(* PLC project Adressering.ecp, WAGO e!COCKPIT e!COCKPIT *)
(* stored: creationDateTime 2021-01-18T14:20:23.2110188, modificationDateTime 2021-01-18T11:51:27.6823754 *)

TYPE dtRomtype_99999 : STRUCT
  RB601_V : BOOL;  (* Bevegelse *)
  RB602_V : BOOL;  (* Bevegelse *)
  RB603_V : BOOL;  (* Bevegelse *)
  RB604_V : BOOL;  (* Bevegelse *)
  RB605_V : BOOL;  (* Bevegelse *)
  RB606_V : BOOL;  (* Bevegelse *)
  RB607_V : BOOL;  (* Bevegelse *)
  RB608_V : BOOL;  (* Bevegelse *)
  RB609_V : BOOL;  (* Bevegelse *)
  RB601_HVAC : BOOL;  (* HVAC signal *)
  RB602_HVAC : BOOL;  (* HVAC signal *)
  RB603_HVAC : BOOL;  (* HVAC signal *)
  RB604_HVAC : BOOL;  (* HVAC signal *)
  RB605_HVAC : BOOL;  (* HVAC signal *)
  RB606_HVAC : BOOL;  (* HVAC signal *)
  RB607_HVAC : BOOL;  (* HVAC signal *)
  RB608_HVAC : BOOL;  (* HVAC signal *)
  RB609_HVAC : BOOL;  (* HVAC signal *)
  RT601_CT : REAL;  (* Rom temperatur *)
  RT602_CT : REAL;  (* Rom temperatur *)
  RT602_SP : REAL;  (* Temperatur SP *)
  RT603_CT : REAL;  (* Rom temperatur *)
  RT603_SP : REAL;  (* Temperatur SP *)
  RT604_CT : REAL;  (* Rom temperatur *)
  RT604_SP : REAL;  (* Temperatur SP *)
  RT605_CT : REAL;  (* Rom temperatur *)
  RT605_SP : REAL;  (* Temperatur SP *)
  RT606_CT : REAL;  (* Rom temperatur *)
  RT606_SP : REAL;  (* Temperatur SP *)
  RT607_CT : REAL;  (* Rom temperatur *)
  RT607_SP : REAL;  (* Temperatur SP *)
  RT608_CT : REAL;  (* Rom temperatur *)
  RT608_SP : REAL;  (* Temperatur SP *)
  RT609_CT : REAL;  (* Rom temperatur *)
  RT609_SP : REAL;  (* Temperatur SP *)
  RT601_SP_D : REAL;  (* Temperatur SP *)
  RT601_SP_S : REAL;  (* Temperatur SP standby *)
  RT601_SP_N : REAL;  (* Temperatur SP nattsenk *)
  RT601_SP_F : REAL;  (* Temperatur SP frostsikring *)
  RT601_CS : REAL;  (* Aktivt temperatur SP *)
  OPM : INT;  (* Rom modus *)
  OPM_CV : INT;  (* Rom modus verdi *)
  RY601_CV : REAL;  (* Co2 Nivaa *)
  RY602_CV : REAL;  (* Co2 Nivaa *)
  RY603_CV : REAL;  (* Co2 Nivaa *)
  RY604_CV : REAL;  (* Co2 Nivaa *)
  RY605_CV : REAL;  (* Co2 Nivaa *)
  RY606_CV : REAL;  (* Co2 Nivaa *)
  RY607_CV : REAL;  (* Co2 Nivaa *)
  RY608_CV : REAL;  (* Co2 Nivaa *)
  RY609_CV : REAL;  (* Co2 Nivaa *)
  RY601_SP : REAL;  (* Co2 SP *)
  RY601_MAN : BOOL;  (* Co2 Man mode *)
  RY601_OP : REAL;  (* Co2 paadrag *)
  LH601_OP : REAL;  (* Varmepaadrag *)
  LH602_OP : REAL;  (* Varmepaadrag *)
  LH603_OP : REAL;  (* Varmepaadrag *)
  LH604_OP : REAL;  (* Varmepaadrag *)
  LH605_OP : REAL;  (* Varmepaadrag *)
  LH606_OP : REAL;  (* Varmepaadrag *)
  LH607_OP : REAL;  (* Varmepaadrag *)
  LH608_OP : REAL;  (* Varmepaadrag *)
  LH609_OP : REAL;  (* Varmepaadrag *)
  LH601_MAN : BOOL;  (* Force LH *)
END_STRUCT;
END_TYPE

TYPE dtRomtype_9992 : STRUCT
  RB601_V : BOOL;  (* Bevegelse *)
  RB602_V : BOOL;  (* Bevegelse *)
  RB603_V : BOOL;  (* Bevegelse *)
  RB604_V : BOOL;  (* Bevegelse *)
  RB605_V : BOOL;  (* Bevegelse *)
  RB606_V : BOOL;  (* Bevegelse *)
  RB607_V : BOOL;  (* Bevegelse *)
  RB608_V : BOOL;  (* Bevegelse *)
  RB609_V : BOOL;  (* Bevegelse *)
  RB601_HVAC : BOOL;  (* HVAC signal *)
  RB602_HVAC : BOOL;  (* HVAC signal *)
  RB603_HVAC : BOOL;  (* HVAC signal *)
  RB604_HVAC : BOOL;  (* HVAC signal *)
  RB605_HVAC : BOOL;  (* HVAC signal *)
  RB606_HVAC : BOOL;  (* HVAC signal *)
  RB607_HVAC : BOOL;  (* HVAC signal *)
  RB608_HVAC : BOOL;  (* HVAC signal *)
  RB609_HVAC : BOOL;  (* HVAC signal *)
  RT601_CT : REAL;  (* Rom temperatur *)
  RT602_CT : REAL;  (* Rom temperatur *)
  RT602_SP : REAL;  (* Temperatur SP *)
  RT603_CT : REAL;  (* Rom temperatur *)
  RT603_SP : REAL;  (* Temperatur SP *)
  RT604_CT : REAL;  (* Rom temperatur *)
  RT604_SP : REAL;  (* Temperatur SP *)
  RT605_CT : REAL;  (* Rom temperatur *)
  RT605_SP : REAL;  (* Temperatur SP *)
  RT606_CT : REAL;  (* Rom temperatur *)
  RT606_SP : REAL;  (* Temperatur SP *)
  RT607_CT : REAL;  (* Rom temperatur *)
  RT607_SP : REAL;  (* Temperatur SP *)
  RT608_CT : REAL;  (* Rom temperatur *)
  RT608_SP : REAL;  (* Temperatur SP *)
  RT609_CT : REAL;  (* Rom temperatur *)
  RT609_SP : REAL;  (* Temperatur SP *)
  RT601_SP_D : REAL;  (* Temperatur SP *)
  RT601_SP_S : REAL;  (* Temperatur SP standby *)
  RT601_SP_N : REAL;  (* Temperatur SP nattsenk *)
  RT601_SP_F : REAL;  (* Temperatur SP frostsikring *)
  RT601_CS : REAL;  (* Aktivt temperatur SP *)
  OPM : INT;  (* Rom modus *)
  OPM_CV : INT;  (* Rom modus verdi *)
  RY601_CV : REAL;  (* Co2 Nivaa *)
  RY602_CV : REAL;  (* Co2 Nivaa *)
  RY601_SP : REAL;  (* Co2 SP *)
  RY601_MAN : BOOL;  (* Co2 Man mode *)
  RY601_OP : REAL;  (* Co2 paadrag *)
END_STRUCT;
END_TYPE

TYPE dtRomtype_111001 : STRUCT
  RB601_V : BOOL;  (* Bevegelse *)
  RB601_HVAC : BOOL;  (* HVAC signal *)
  RT601_CT : REAL;  (* Rom temperatur *)
  RT601_SP_D : REAL;  (* Temperatur SP *)
  RT601_SP_S : REAL;  (* Temperatur SP standby *)
  RT601_SP_N : REAL;  (* Temperatur SP nattsenk *)
  RT601_SP_F : REAL;  (* Temperatur SP frostsikring *)
  RT601_CS : REAL;  (* Aktivt temperatur SP *)
  OPM : INT;  (* Rom modus *)
  OPM_CV : INT;  (* Rom modus verdi *)
  LH601_CMD : BOOL;  (* LH601_CMD *)
  LH601_MAN : BOOL;  (* Force LH *)
END_STRUCT;
END_TYPE

TYPE dtRomtype_111111111111111 : STRUCT
  RB601_V : BOOL;  (* Bevegelse *)
  RB601_HVAC : BOOL;  (* HVAC signal *)
  RT601_CT : REAL;  (* Rom temperatur *)
  RT601_SP_D : REAL;  (* Temperatur SP *)
  RT601_SP_S : REAL;  (* Temperatur SP standby *)
  RT601_SP_N : REAL;  (* Temperatur SP nattsenk *)
  RT601_SP_F : REAL;  (* Temperatur SP frostsikring *)
  RT601_CS : REAL;  (* Aktivt temperatur SP *)
  OPM : INT;  (* Rom modus *)
  OPM_CV : INT;  (* Rom modus verdi *)
  RY601_CV : REAL;  (* Co2 Nivaa *)
  RY601_SP : REAL;  (* Co2 SP *)
  RY601_MAN : BOOL;  (* Co2 Man mode *)
  RY601_OP : REAL;  (* Co2 paadrag *)
  LH601_OP : REAL;  (* Varmepaadrag *)
  LH601_MAN : BOOL;  (* Force LH *)
  LH601_CMD : BOOL;  (* LH601_CMD *)
  LC601_OP : REAL;  (* LC601_OP *)
  LC601_SP : REAL;  (* LC SP *)
  LC601_MAN : BOOL;  (* Force LC *)
  LC601_CMD : BOOL;  (* LC601_CMD *)
  RT601_SP : REAL;  (* Temperatur SP feedback *)
  RT601_SP_FB : REAL;  (* Temperatur SP *)
  RT601_SP_IN : REAL;  (* Temperatur SP lokalt panel *)
  LU601_V : BOOL;  (* Befukter status *)
  LU601_AL : BOOL;  (* Befukter alarm/feil *)
  LU601_CMD : BOOL;  (* Befukter tillat start *)
  OPM_001 : BYTE;  (* OPM output *)
  RH601 : REAL;  (* Rom fuktighet *)
END_STRUCT;
END_TYPE

{attribute 'qualified_only'}
VAR_GLOBAL  (* STLV59_563 *)
  STLV59_A_563_RB001_HVAC : BOOL;  (* HVAC signal for PLS *)
  STLV59_A_563_KNX_Card_1_Status : BOOL;  (* KNX kort 1 status *)
  STLV59_A_563_001 : dtRomtype_99999;  (* Placeholder 1 *)
  STLV59_A_563_002 : dtRomtype_99999;  (* Placeholder 2 *)
  STLV59_A_563_003 : dtRomtype_9992;  (* Placeholder 3 *)
  STLV59_A_563_4K302 : dtRomtype_111001;  (* Herre garderobe *)
  STLV59_A_563_4L302 : dtRomtype_111001;  (* Dame garderobe *)
  STLV59_A_563_4H201 : dtRomtype_111111111111111;  (* test *)
END_VAR

FUNCTION_BLOCK fbRomtype_99999
  VAR_INPUT
    RB601_HVAC : BOOL;
    RB602_HVAC : BOOL;
    RB603_HVAC : BOOL;
    RB604_HVAC : BOOL;
    RB605_HVAC : BOOL;
    RB606_HVAC : BOOL;
    RB607_HVAC : BOOL;
    RB608_HVAC : BOOL;
    RB609_HVAC : BOOL;
    RT601_CT : REAL;
    RT602_CT : REAL;
    RT602_SP : REAL;
    RT603_CT : REAL;
    RT603_SP : REAL;
    RT604_CT : REAL;
    RT604_SP : REAL;
    RT605_CT : REAL;
    RT605_SP : REAL;
    RT606_CT : REAL;
    RT606_SP : REAL;
    RT607_CT : REAL;
    RT607_SP : REAL;
    RT608_CT : REAL;
    RT608_SP : REAL;
    RT609_CT : REAL;
    RT609_SP : REAL;
    RT601_SP_D : REAL;
    RT601_SP_S : REAL;
    RT601_SP_N : REAL;
    RT601_SP_F : REAL;
    OPM : INT;
    RY601_CV : REAL;
    RY602_CV : REAL;
    RY603_CV : REAL;
    RY604_CV : REAL;
    RY605_CV : REAL;
    RY606_CV : REAL;
    RY607_CV : REAL;
    RY608_CV : REAL;
    RY609_CV : REAL;
    RY601_SP : REAL;
    RY601_MAN : BOOL;
    LH601_MAN : BOOL;
  END_VAR
  VAR_OUTPUT
    OPM_CV : INT;
    RT601_CS : REAL;
    RT602_CS : REAL;
    RT603_CS : REAL;
    RT604_CS : REAL;
    RT605_CS : REAL;
    RT606_CS : REAL;
    RT607_CS : REAL;
    RT608_CS : REAL;
    RT609_CS : REAL;
    RY601_OP : REAL;
    RY602_OP : REAL;
    RY603_OP : REAL;
    RY604_OP : REAL;
    RY605_OP : REAL;
    RY606_OP : REAL;
    RY607_OP : REAL;
    RY608_OP : REAL;
    RY609_OP : REAL;
    LH601_OP : REAL;
    LH602_OP : REAL;
    LH603_OP : REAL;
    LH604_OP : REAL;
    LH605_OP : REAL;
    LH606_OP : REAL;
    LH607_OP : REAL;
    LH608_OP : REAL;
    LH609_OP : REAL;
  END_VAR

(* CFC diagram, written out as Structured Text *)
END_FUNCTION_BLOCK

FUNCTION_BLOCK fbRomtype_9992
  VAR_INPUT
    RB601_HVAC : BOOL;
    RB602_HVAC : BOOL;
    RB603_HVAC : BOOL;
    RB604_HVAC : BOOL;
    RB605_HVAC : BOOL;
    RB606_HVAC : BOOL;
    RB607_HVAC : BOOL;
    RB608_HVAC : BOOL;
    RB609_HVAC : BOOL;
    RT601_CT : REAL;
    RT602_CT : REAL;
    RT602_SP : REAL;
    RT603_CT : REAL;
    RT603_SP : REAL;
    RT604_CT : REAL;
    RT604_SP : REAL;
    RT605_CT : REAL;
    RT605_SP : REAL;
    RT606_CT : REAL;
    RT606_SP : REAL;
    RT607_CT : REAL;
    RT607_SP : REAL;
    RT608_CT : REAL;
    RT608_SP : REAL;
    RT609_CT : REAL;
    RT609_SP : REAL;
    RT601_SP_D : REAL;
    RT601_SP_S : REAL;
    RT601_SP_N : REAL;
    RT601_SP_F : REAL;
    OPM : INT;
    RY601_CV : REAL;
    RY602_CV : REAL;
    RY601_SP : REAL;
    RY601_MAN : BOOL;
  END_VAR
  VAR_OUTPUT
    OPM_CV : INT;
    RT601_CS : REAL;
    RT602_CS : REAL;
    RT603_CS : REAL;
    RT604_CS : REAL;
    RT605_CS : REAL;
    RT606_CS : REAL;
    RT607_CS : REAL;
    RT608_CS : REAL;
    RT609_CS : REAL;
    RY601_OP : REAL;
    RY602_OP : REAL;
  END_VAR

(* CFC diagram, written out as Structured Text *)
END_FUNCTION_BLOCK

FUNCTION_BLOCK fbRomtype_111001
  VAR_INPUT
    RB601_HVAC : BOOL;
    RT601_CT : REAL;
    RT601_SP_D : REAL;
    RT601_SP_S : REAL;
    RT601_SP_N : REAL;
    RT601_SP_F : REAL;
    OPM : INT;
    LH601_MAN : BOOL;
  END_VAR
  VAR_OUTPUT
    OPM_CV : INT;
    RT601_CS : REAL;
    LH601_CMD : BOOL;
  END_VAR

(* CFC diagram, written out as Structured Text *)
END_FUNCTION_BLOCK

FUNCTION_BLOCK fbRomtype_111111111111111
  VAR_INPUT
    RB601_HVAC : BOOL;
    RT601_CT : REAL;
    RT601_SP_D : REAL;
    RT601_SP_S : REAL;
    RT601_SP_N : REAL;
    RT601_SP_F : REAL;
    OPM : INT;
    RY601_CV : REAL;
    RY601_SP : REAL;
    RY601_MAN : BOOL;
    LH601_MAN : BOOL;
    LC601_SP : REAL;
    LC601_MAN : BOOL;
    RT601_SP_IN : REAL;
    LU601_V : BOOL;
    RH601_CV : REAL;
  END_VAR
  VAR_OUTPUT
    OPM_CV : INT;
    RT601_CS : REAL;
    RY601_OP : REAL;
    LH601_OP : REAL;
    LH601_CMD : BOOL;
    LC601_OP : REAL;
    LC601_CMD : BOOL;
    LU601_CMD : BOOL;
    OPM_001 : BYTE;
  END_VAR

(* CFC diagram, written out as Structured Text *)
END_FUNCTION_BLOCK

FUNCTION_BLOCK fbSE_Hyst
  VAR_INPUT
    rIn : REAL;
    rOn : REAL;
    rOff : REAL;
  END_VAR
  VAR_OUTPUT
    xOut : BOOL;
  END_VAR

					xOut:= ((rOn > rOff AND (rIn >= rOn OR (xOut AND rIn > rOff)))	OR		(rOn <rOff AND (rIn <= rOn OR (xOut AND rIn <rOff))));
				
END_FUNCTION_BLOCK

FUNCTION_BLOCK fbSE_PID
  VAR_INPUT
    ifPv : REAL;  (* Prosessvariabel (actual) *)
    ifSp : REAL;  (* Settpunkt *)
    ifKp : REAL := 1;  (* Forsterkning *)
    ifTi : REAL := 10;  (* I-tid *)
    ifTd : REAL;  (* D-tid *)
    ifBias : REAL;  (* Bias (Statisk paadrag som alltid er der) 0-100% *)
    ifInZero : REAL;  (* Nullpunkt for inn-verdi (PV og SP) *)
    ifInMax : REAL := 100;  (* Toppunkt for inn-verdi (PV og SP) *)
    ifOutZero : REAL;  (* Nullpunkt for ut-verdi (MV) *)
    ifOutMax : REAL := 100;  (* Toppunkt for ut-verdi (MV) *)
    ixManMode : BOOL;  (* Sender ManMv som MV, og resetter I-ledd *)
    ifManMv : REAL;  (* Manuelt paadrag som brukes i Man mode *)
  END_VAR
  VAR
    fPv : REAL;  (* Skalert PV (0-100) *)
    fSp : REAL;  (* Skalert SP (0-100) *)
    eRun : R_TRIG;  (* Resetter I-ledd ved endring rising edge i start betingelser *)
    fAvvik : REAL;  (* Avvik (Error) *)
    tCycleTimer : TON := (PT := TIME#1s0ms);  (* Teller syklus tiden *)
    fCycleTime : REAL;  (* Syklus tid i real *)
    fPID : REAL;  (* PID resultat (0-100%) *)
    fLastKp : REAL;  (* Forsterkning sist syklus (brukes til skalering ved endring) *)
    fLastTi : REAL;  (* Ti sist syklus (brukes til skalering ved endring) *)
    fLastIntegMax : REAL;  (* Max integral verdi sist syklus *)
    fIntegMax : REAL;  (* Max integral verdi (beregnet med Ti) *)
    fIntegral : REAL;  (* Integral verdi *)
    fI : REAL;  (* Integralt avvik *)
    fLastAvvik : REAL;  (* Avvik sist syklus *)
    fDerivat : REAL;  (* Derivat verdi *)
    fD : REAL;  (* Derivert avvik *)
  END_VAR
  VAR_OUTPUT
    qfMv : REAL;  (* Manipulert verdi (Resultat av PID) *)
    qxError : BOOL;  (* Feil alarm *)
  END_VAR

					eRun(CLK:= (ifKp > 0 AND NOT ixManMode));

IF ixManMode THEN																//Skriver manuelt SP til utgang
	qfMv := ifManMv;
ELSIF eRun.Q THEN																//Hvis det er rising edge paastart betingelser vil diverse variabler resettes/initializes
	fIntegral := 0;
	fIntegMax:= fLastIntegMax := 1 / ifKp * (100 / (1 / ifTi));
	fLastTi:= ifTi;
	fLastKp:= ifKp;
	fLastAvvik:= fAvvik;
	tCycleTimer(IN:= FALSE);
	tCycleTimer(IN:= TRUE);
ELSIF ifKp > 0 THEN												//Hvis Kp er satt, kjoeres PID funksjon

	//Felles
		IF(ifInMax - ifInZero) = 0 THEN											//Sjekker om vi deler paa 0, og gir ut evt. feil
		qxError := TRUE;
		RETURN;
	ELSE																		//	Ellers omskaleres Inn-verdier fra valgt til 0-100, og feil resettes
		qxError := FALSE;
		fPv:= (100 / (ifInMax - ifInZero)) * (ifPv - ifInZero);
		fSp:= (100 / (ifInMax - ifInZero)) * (ifSP - ifInZero);
	END_IF

	//Teller syklys tid
	tCycleTimer();																//Kjoerer TON for aa sjekke hvor lang tid som har gaatt siden forgje utregning
	fCycleTime:= 0.001 * TIME_TO_REAL(tCycleTimer.ET);							//Omskalerer syklus tid fra TIME til REAL
	tCycleTimer(IN:= FALSE);													//Resetter TON
	tCycleTimer(IN:= TRUE);


	//Proporsjonalt avvik
	fAvvik:= fSp - fPv;															//Beregner avvik som brukes i P-leddet


	//Integralt avvik
	IF ifTi > 0 THEN															//Hvis I er mer en 0, kjoerer vi I-ledd beregning
		IF ifTi <> fLastTi OR ifKp <> fLastKp THEN								//Hvis Ti eller Kp endrer seg, omskaleres max verdi for integral og den eksisterende integral verdien. Lagrer div variabler til neste sjekk/skalering
			fIntegMax := 1 / ifKp * (100 / (1 / ifTi));
			fIntegral:= (fIntegMax / fLastIntegMax) * fIntegral;
			fLastIntegMax:= fIntegMax;
			fLastTi:= ifTi;
			fLastKp:= ifKp;
		END_IF

		fIntegral := LIMIT(0, (fIntegral + fAvvik * fCycleTime), fIntegMax);		//Beregner integral

		fI:= (1 / ifTi) * fIntegral;												//Beregner I-verdien

	ELSE
		fI := 0;																	//Skriver i til 0 hvis Ti er 0
	END_IF

	//Derivert avvik
	IF(fAvvik - fLastAvvik)<> 0  AND ifTd > 0 THEN							//Sjekker om D-ledd er i bruk, og hindrer at vi deler paa 0 ved feil
		fDerivat := (fAvvik - fLastAvvik) / fCycleTime;							//Deriverer avviket
		fD:= LIMIT(-100, (ifTd * fDerivat), 100);								//Beregner D-verdien
	ELSE
		fD := 0;
	END_IF


	//PID utregnign
	fPID:= LIMIT(0, (ifKp * (fAvvik + fI + fD) + ifBias), 100);				//Beregner PID utverdi i 0-100

	IF(ifOutMax - ifOutZero) = 0 THEN											//Sjekker om vi deler paa 0
		qxError := TRUE;
	ELSE																		//	Hvis ikke, omskaleres ut signal til valgt span og feil resettes
		qxError := FALSE;
		qfMv:= ((ifOutMax - ifOutZero) / 100) * fPID + ifOutZero;
	END_IF

ELSE																			//Skriver utgang til 0, hvis PID ikke er paa
	qfMv := 0;
END_IF
				
END_FUNCTION_BLOCK

PROGRAM PRG_KNX_563_1
  VAR
    i : INT := 0;  (* Felles *)
    Interval : TON := (PT := TIME#2m0s0ms);
    typDPT : typDPT;
    KNX_master_1 : WagoAppKNX.FbKNX_Master;  (* Master *)
    M1_001_001_RB601_V : fbDPT_Switch_pro;  (* 001 *)
    M1_002_001_RB602_V : fbDPT_Switch_pro;
    M1_003_001_RB603_V : fbDPT_Switch_pro;
    M1_004_001_RB604_V : fbDPT_Switch_pro;
    M1_005_001_RB605_V : fbDPT_Switch_pro;
    M1_006_001_RB606_V : fbDPT_Switch_pro;
    M1_007_001_RB607_V : fbDPT_Switch_pro;
    M1_008_001_RB608_V : fbDPT_Switch_pro;
    M1_009_001_RB609_V : fbDPT_Switch_pro;
    M1_010_001_RB601_HVAC : fbDPT_Switch_pro;
    M1_011_001_RB602_HVAC : fbDPT_Switch_pro;
    M1_012_001_RB603_HVAC : fbDPT_Switch_pro;
    M1_013_001_RB604_HVAC : fbDPT_Switch_pro;
    M1_014_001_RB605_HVAC : fbDPT_Switch_pro;
    M1_015_001_RB606_HVAC : fbDPT_Switch_pro;
    M1_016_001_RB607_HVAC : fbDPT_Switch_pro;
    M1_017_001_RB608_HVAC : fbDPT_Switch_pro;
    M1_018_001_RB609_HVAC : fbDPT_Switch_pro;
    M1_019_001_RT601_CT : fbDPT_Value_Temp_pro;
    M1_020_001_RT602_CT : fbDPT_Value_Temp_pro;
    M1_021_001_RT603_CT : fbDPT_Value_Temp_pro;
    M1_022_001_RT604_CT : fbDPT_Value_Temp_pro;
    M1_023_001_RT605_CT : fbDPT_Value_Temp_pro;
    M1_024_001_RT606_CT : fbDPT_Value_Temp_pro;
    M1_025_001_RT607_CT : fbDPT_Value_Temp_pro;
    M1_026_001_RT608_CT : fbDPT_Value_Temp_pro;
    M1_027_001_RT609_CT : fbDPT_Value_Temp_pro;
    M1_028_001_RY601_CV : fbDPT_Value_AirQuality_pro;
    M1_029_001_RY602_CV : fbDPT_Value_AirQuality_pro;
    M1_030_001_RY603_CV : fbDPT_Value_AirQuality_pro;
    M1_031_001_RY604_CV : fbDPT_Value_AirQuality_pro;
    M1_032_001_RY605_CV : fbDPT_Value_AirQuality_pro;
    M1_033_001_RY606_CV : fbDPT_Value_AirQuality_pro;
    M1_034_001_RY607_CV : fbDPT_Value_AirQuality_pro;
    M1_035_001_RY608_CV : fbDPT_Value_AirQuality_pro;
    M1_036_001_RY609_CV : fbDPT_Value_AirQuality_pro;
    M1_037_001_LH601_OP : fbDPT_Scaling_pro;
    M1_038_001_LH602_OP : fbDPT_Scaling_pro;
    M1_039_001_LH603_OP : fbDPT_Scaling_pro;
    M1_040_001_LH604_OP : fbDPT_Scaling_pro;
    M1_041_001_LH605_OP : fbDPT_Scaling_pro;
    M1_042_001_LH606_OP : fbDPT_Scaling_pro;
    M1_043_001_LH607_OP : fbDPT_Scaling_pro;
    M1_044_001_LH608_OP : fbDPT_Scaling_pro;
    M1_045_001_LH609_OP : fbDPT_Scaling_pro;
    M1_046_002_RB601_V : fbDPT_Switch_pro;  (* 002 *)
    M1_047_002_RB602_V : fbDPT_Switch_pro;
    M1_048_002_RB603_V : fbDPT_Switch_pro;
    M1_049_002_RB604_V : fbDPT_Switch_pro;
    M1_050_002_RB605_V : fbDPT_Switch_pro;
    M1_051_002_RB606_V : fbDPT_Switch_pro;
    M1_052_002_RB607_V : fbDPT_Switch_pro;
    M1_053_002_RB608_V : fbDPT_Switch_pro;
    M1_054_002_RB609_V : fbDPT_Switch_pro;
    M1_055_002_RB601_HVAC : fbDPT_Switch_pro;
    M1_056_002_RB602_HVAC : fbDPT_Switch_pro;
    M1_057_002_RB603_HVAC : fbDPT_Switch_pro;
    M1_058_002_RB604_HVAC : fbDPT_Switch_pro;
    M1_059_002_RB605_HVAC : fbDPT_Switch_pro;
    M1_060_002_RB606_HVAC : fbDPT_Switch_pro;
    M1_061_002_RB607_HVAC : fbDPT_Switch_pro;
    M1_062_002_RB608_HVAC : fbDPT_Switch_pro;
    M1_063_002_RB609_HVAC : fbDPT_Switch_pro;
    M1_064_002_RT601_CT : fbDPT_Value_Temp_pro;
    M1_065_002_RT602_CT : fbDPT_Value_Temp_pro;
    M1_066_002_RT603_CT : fbDPT_Value_Temp_pro;
    M1_067_002_RT604_CT : fbDPT_Value_Temp_pro;
    M1_068_002_RT605_CT : fbDPT_Value_Temp_pro;
    M1_069_002_RT606_CT : fbDPT_Value_Temp_pro;
    M1_070_002_RT607_CT : fbDPT_Value_Temp_pro;
    M1_071_002_RT608_CT : fbDPT_Value_Temp_pro;
    M1_072_002_RT609_CT : fbDPT_Value_Temp_pro;
    M1_073_002_RY601_CV : fbDPT_Value_AirQuality_pro;
    M1_074_002_RY602_CV : fbDPT_Value_AirQuality_pro;
    M1_075_002_RY603_CV : fbDPT_Value_AirQuality_pro;
    M1_076_002_RY604_CV : fbDPT_Value_AirQuality_pro;
    M1_077_002_RY605_CV : fbDPT_Value_AirQuality_pro;
    M1_078_002_RY606_CV : fbDPT_Value_AirQuality_pro;
    M1_079_002_RY607_CV : fbDPT_Value_AirQuality_pro;
    M1_080_002_RY608_CV : fbDPT_Value_AirQuality_pro;
    M1_081_002_RY609_CV : fbDPT_Value_AirQuality_pro;
    M1_082_002_LH601_OP : fbDPT_Scaling_pro;
    M1_083_002_LH602_OP : fbDPT_Scaling_pro;
    M1_084_002_LH603_OP : fbDPT_Scaling_pro;
    M1_085_002_LH604_OP : fbDPT_Scaling_pro;
    M1_086_002_LH605_OP : fbDPT_Scaling_pro;
    M1_087_002_LH606_OP : fbDPT_Scaling_pro;
    M1_088_002_LH607_OP : fbDPT_Scaling_pro;
    M1_089_002_LH608_OP : fbDPT_Scaling_pro;
    M1_090_002_LH609_OP : fbDPT_Scaling_pro;
    M1_091_003_RB601_V : fbDPT_Switch_pro;  (* 003 *)
    M1_092_003_RB602_V : fbDPT_Switch_pro;
    M1_093_003_RB603_V : fbDPT_Switch_pro;
    M1_094_003_RB604_V : fbDPT_Switch_pro;
    M1_095_003_RB605_V : fbDPT_Switch_pro;
    M1_096_003_RB606_V : fbDPT_Switch_pro;
    M1_097_003_RB607_V : fbDPT_Switch_pro;
    M1_098_003_RB608_V : fbDPT_Switch_pro;
    M1_099_003_RB609_V : fbDPT_Switch_pro;
    M1_100_003_RB601_HVAC : fbDPT_Switch_pro;
    M1_101_003_RB602_HVAC : fbDPT_Switch_pro;
    M1_102_003_RB603_HVAC : fbDPT_Switch_pro;
    M1_103_003_RB604_HVAC : fbDPT_Switch_pro;
    M1_104_003_RB605_HVAC : fbDPT_Switch_pro;
    M1_105_003_RB606_HVAC : fbDPT_Switch_pro;
    M1_106_003_RB607_HVAC : fbDPT_Switch_pro;
    M1_107_003_RB608_HVAC : fbDPT_Switch_pro;
    M1_108_003_RB609_HVAC : fbDPT_Switch_pro;
    M1_109_003_RT601_CT : fbDPT_Value_Temp_pro;
    M1_110_003_RT602_CT : fbDPT_Value_Temp_pro;
    M1_111_003_RT603_CT : fbDPT_Value_Temp_pro;
    M1_112_003_RT604_CT : fbDPT_Value_Temp_pro;
    M1_113_003_RT605_CT : fbDPT_Value_Temp_pro;
    M1_114_003_RT606_CT : fbDPT_Value_Temp_pro;
    M1_115_003_RT607_CT : fbDPT_Value_Temp_pro;
    M1_116_003_RT608_CT : fbDPT_Value_Temp_pro;
    M1_117_003_RT609_CT : fbDPT_Value_Temp_pro;
    M1_118_003_RY601_CV : fbDPT_Value_AirQuality_pro;
    M1_119_003_RY602_CV : fbDPT_Value_AirQuality_pro;
    M1_120_4K302_RB601_V : fbDPT_Switch_pro;  (* 4K302 *)
    M1_121_4K302_RB601_HVAC : fbDPT_Switch_pro;
    M1_122_4K302_RT601_CT : fbDPT_Value_Temp_pro;
    M1_123_4K302_LH601_CMD : fbDPT_Switch_pro;
    M1_124_4L302_RB601_V : fbDPT_Switch_pro;  (* 4L302 *)
    M1_125_4L302_RB601_HVAC : fbDPT_Switch_pro;
    M1_126_4L302_RT601_CT : fbDPT_Value_Temp_pro;
    M1_127_4L302_LH601_CMD : fbDPT_Switch_pro;
    M1_128_4H201_RB601_V : fbDPT_Switch_pro;  (* 4H201 *)
    M1_129_4H201_RB601_HVAC : fbDPT_Switch_pro;
    M1_130_4H201_RT601_CT : fbDPT_Value_Temp_pro;
    M1_131_4H201_RY601_CV : fbDPT_Value_AirQuality_pro;
    M1_132_4H201_LH601_OP : fbDPT_Scaling_pro;
    M1_133_4H201_LH601_CMD : fbDPT_Switch_pro;
    M1_134_4H201_LC601_OP : fbDPT_Scaling_pro;
    M1_135_4H201_LC601_CMD : fbDPT_Switch_pro;
    M1_136_4H201_RT601_SP : fbDPT_Value_Temp_pro;
    M1_137_4H201_RT601_SP_FB : fbDPT_Value_Temp_pro;
    M1_138_4H201_LU601_V : fbDPT_Switch_pro;
    M1_139_4H201_LU601_AL : fbDPT_Switch_pro;
    M1_140_4H201_LU601_CMD : fbDPT_Switch_pro;
    M1_141_4H201_OPM_001 : fbDPT_1_BYTE;
    M1_142_4H201_RH601_CV : FbDPT_Value_Humidity_pro;
  END_VAR
  VAR  (* added by the conversion: wires and edge detectors of the diagram *)
    _ADD9_OUT : INT;
    _GT15_OUT : BOOL;
    _MOVE19_ENO : BOOL;
    _MOVE19_OUT : INT;
    _MOVE46_ENO : BOOL;
    _MOVE46_OUT : ANY;
    _MOVE59_ENO : BOOL;
    _MOVE59_OUT : ANY;
    _MOVE72_ENO : BOOL;
    _MOVE72_OUT : ANY;
    _MOVE85_ENO : BOOL;
    _MOVE85_OUT : ANY;
    _MOVE98_ENO : BOOL;
    _MOVE98_OUT : ANY;
    _MOVE111_ENO : BOOL;
    _MOVE111_OUT : ANY;
    _MOVE124_ENO : BOOL;
    _MOVE124_OUT : ANY;
    _MOVE137_ENO : BOOL;
    _MOVE137_OUT : ANY;
    _MOVE150_ENO : BOOL;
    _MOVE150_OUT : ANY;
    _MOVE163_ENO : BOOL;
    _MOVE163_OUT : ANY;
    _MOVE176_ENO : BOOL;
    _MOVE176_OUT : ANY;
    _MOVE189_ENO : BOOL;
    _MOVE189_OUT : ANY;
    _MOVE202_ENO : BOOL;
    _MOVE202_OUT : ANY;
    _MOVE215_ENO : BOOL;
    _MOVE215_OUT : ANY;
    _MOVE228_ENO : BOOL;
    _MOVE228_OUT : ANY;
    _MOVE241_ENO : BOOL;
    _MOVE241_OUT : ANY;
    _MOVE254_ENO : BOOL;
    _MOVE254_OUT : ANY;
    _MOVE267_ENO : BOOL;
    _MOVE267_OUT : ANY;
    _MOVE280_ENO : BOOL;
    _MOVE280_OUT : ANY;
    _MOVE293_ENO : BOOL;
    _MOVE293_OUT : ANY;
    _MOVE306_ENO : BOOL;
    _MOVE306_OUT : ANY;
    _MOVE319_ENO : BOOL;
    _MOVE319_OUT : ANY;
    _MOVE332_ENO : BOOL;
    _MOVE332_OUT : ANY;
    _MOVE345_ENO : BOOL;
    _MOVE345_OUT : ANY;
    _MOVE358_ENO : BOOL;
    _MOVE358_OUT : ANY;
    _MOVE371_ENO : BOOL;
    _MOVE371_OUT : ANY;
    _MOVE384_ENO : BOOL;
    _MOVE384_OUT : ANY;
    _MOVE397_ENO : BOOL;
    _MOVE397_OUT : ANY;
    _MOVE410_ENO : BOOL;
    _MOVE410_OUT : ANY;
    _MOVE423_ENO : BOOL;
    _MOVE423_OUT : ANY;
    _MOVE436_ENO : BOOL;
    _MOVE436_OUT : ANY;
    _MOVE449_ENO : BOOL;
    _MOVE449_OUT : ANY;
    _MOVE462_ENO : BOOL;
    _MOVE462_OUT : ANY;
    _MOVE475_ENO : BOOL;
    _MOVE475_OUT : ANY;
    _MOVE488_ENO : BOOL;
    _MOVE488_OUT : ANY;
    _MOVE501_ENO : BOOL;
    _MOVE501_OUT : ANY;
    _MOVE659_ENO : BOOL;
    _MOVE659_OUT : ANY;
    _MOVE672_ENO : BOOL;
    _MOVE672_OUT : ANY;
    _MOVE685_ENO : BOOL;
    _MOVE685_OUT : ANY;
    _MOVE698_ENO : BOOL;
    _MOVE698_OUT : ANY;
    _MOVE711_ENO : BOOL;
    _MOVE711_OUT : ANY;
    _MOVE724_ENO : BOOL;
    _MOVE724_OUT : ANY;
    _MOVE737_ENO : BOOL;
    _MOVE737_OUT : ANY;
    _MOVE750_ENO : BOOL;
    _MOVE750_OUT : ANY;
    _MOVE763_ENO : BOOL;
    _MOVE763_OUT : ANY;
    _MOVE776_ENO : BOOL;
    _MOVE776_OUT : ANY;
    _MOVE789_ENO : BOOL;
    _MOVE789_OUT : ANY;
    _MOVE802_ENO : BOOL;
    _MOVE802_OUT : ANY;
    _MOVE815_ENO : BOOL;
    _MOVE815_OUT : ANY;
    _MOVE828_ENO : BOOL;
    _MOVE828_OUT : ANY;
    _MOVE841_ENO : BOOL;
    _MOVE841_OUT : ANY;
    _MOVE854_ENO : BOOL;
    _MOVE854_OUT : ANY;
    _MOVE867_ENO : BOOL;
    _MOVE867_OUT : ANY;
    _MOVE880_ENO : BOOL;
    _MOVE880_OUT : ANY;
    _MOVE893_ENO : BOOL;
    _MOVE893_OUT : ANY;
    _MOVE906_ENO : BOOL;
    _MOVE906_OUT : ANY;
    _MOVE919_ENO : BOOL;
    _MOVE919_OUT : ANY;
    _MOVE932_ENO : BOOL;
    _MOVE932_OUT : ANY;
    _MOVE945_ENO : BOOL;
    _MOVE945_OUT : ANY;
    _MOVE958_ENO : BOOL;
    _MOVE958_OUT : ANY;
    _MOVE971_ENO : BOOL;
    _MOVE971_OUT : ANY;
    _MOVE984_ENO : BOOL;
    _MOVE984_OUT : ANY;
    _MOVE997_ENO : BOOL;
    _MOVE997_OUT : ANY;
    _MOVE1010_ENO : BOOL;
    _MOVE1010_OUT : ANY;
    _MOVE1023_ENO : BOOL;
    _MOVE1023_OUT : ANY;
    _MOVE1036_ENO : BOOL;
    _MOVE1036_OUT : ANY;
    _MOVE1049_ENO : BOOL;
    _MOVE1049_OUT : ANY;
    _MOVE1062_ENO : BOOL;
    _MOVE1062_OUT : ANY;
    _MOVE1075_ENO : BOOL;
    _MOVE1075_OUT : ANY;
    _MOVE1088_ENO : BOOL;
    _MOVE1088_OUT : ANY;
    _MOVE1101_ENO : BOOL;
    _MOVE1101_OUT : ANY;
    _MOVE1114_ENO : BOOL;
    _MOVE1114_OUT : ANY;
    _MOVE1272_ENO : BOOL;
    _MOVE1272_OUT : ANY;
    _MOVE1285_ENO : BOOL;
    _MOVE1285_OUT : ANY;
    _MOVE1298_ENO : BOOL;
    _MOVE1298_OUT : ANY;
    _MOVE1311_ENO : BOOL;
    _MOVE1311_OUT : ANY;
    _MOVE1324_ENO : BOOL;
    _MOVE1324_OUT : ANY;
    _MOVE1337_ENO : BOOL;
    _MOVE1337_OUT : ANY;
    _MOVE1350_ENO : BOOL;
    _MOVE1350_OUT : ANY;
    _MOVE1363_ENO : BOOL;
    _MOVE1363_OUT : ANY;
    _MOVE1376_ENO : BOOL;
    _MOVE1376_OUT : ANY;
    _MOVE1389_ENO : BOOL;
    _MOVE1389_OUT : ANY;
    _MOVE1402_ENO : BOOL;
    _MOVE1402_OUT : ANY;
    _MOVE1415_ENO : BOOL;
    _MOVE1415_OUT : ANY;
    _MOVE1428_ENO : BOOL;
    _MOVE1428_OUT : ANY;
    _MOVE1441_ENO : BOOL;
    _MOVE1441_OUT : ANY;
    _MOVE1454_ENO : BOOL;
    _MOVE1454_OUT : ANY;
    _MOVE1467_ENO : BOOL;
    _MOVE1467_OUT : ANY;
    _MOVE1480_ENO : BOOL;
    _MOVE1480_OUT : ANY;
    _MOVE1493_ENO : BOOL;
    _MOVE1493_OUT : ANY;
    _MOVE1506_ENO : BOOL;
    _MOVE1506_OUT : ANY;
    _MOVE1519_ENO : BOOL;
    _MOVE1519_OUT : ANY;
    _MOVE1532_ENO : BOOL;
    _MOVE1532_OUT : ANY;
    _MOVE1545_ENO : BOOL;
    _MOVE1545_OUT : ANY;
    _MOVE1558_ENO : BOOL;
    _MOVE1558_OUT : ANY;
    _MOVE1571_ENO : BOOL;
    _MOVE1571_OUT : ANY;
    _MOVE1584_ENO : BOOL;
    _MOVE1584_OUT : ANY;
    _MOVE1597_ENO : BOOL;
    _MOVE1597_OUT : ANY;
    _MOVE1610_ENO : BOOL;
    _MOVE1610_OUT : ANY;
    _MOVE1623_ENO : BOOL;
    _MOVE1623_OUT : ANY;
    _MOVE1636_ENO : BOOL;
    _MOVE1636_OUT : ANY;
    _MOVE1650_ENO : BOOL;
    _MOVE1650_OUT : ANY;
    _MOVE1663_ENO : BOOL;
    _MOVE1663_OUT : ANY;
    _MOVE1676_ENO : BOOL;
    _MOVE1676_OUT : ANY;
    _MOVE1706_ENO : BOOL;
    _MOVE1706_OUT : ANY;
    _MOVE1719_ENO : BOOL;
    _MOVE1719_OUT : ANY;
    _MOVE1732_ENO : BOOL;
    _MOVE1732_OUT : ANY;
    _MOVE1762_ENO : BOOL;
    _MOVE1762_OUT : ANY;
    _MOVE1775_ENO : BOOL;
    _MOVE1775_OUT : ANY;
    _MOVE1788_ENO : BOOL;
    _MOVE1788_OUT : ANY;
    _MOVE1801_ENO : BOOL;
    _MOVE1801_OUT : ANY;
    _MOVE1890_ENO : BOOL;
    _MOVE1890_OUT : ANY;
    _MOVE1903_ENO : BOOL;
    _MOVE1903_OUT : ANY;
    _MOVE1916_ENO : BOOL;
    _MOVE1916_OUT : ANY;
    _MOVE1961_ENO : BOOL;
    _MOVE1961_OUT : ANY;
  END_VAR

(* CFC diagram, written out as Structured Text *)
(* KNX Sending interval *)
(* KNX Master *)
Interval(IN := Interval.Q);
_ADD9_OUT := BOOL_TO_INT(Interval.Q) + i;
i := _ADD9_OUT;
_GT15_OUT := i > 26;
_MOVE19_OUT := MOVE(EN := _GT15_OUT, IN := 0, ENO => _MOVE19_ENO);
IF _MOVE19_ENO THEN i := _MOVE19_OUT; END_IF;
KNX_master_1(I_Port := IoConfig_Globals.KNX_EIB_TP1_Interface, bPortKNX := 1);
STLV59_563.STLV59_A_563_KNX_Card_1_Status := KNX_master_1.sStatus = 'OK';
(* Rom 001 *)
(* RB601_V *)
(* RB602_V *)
M1_001_001_RB601_V(bPortKNX := 1, dwIndex_DPT := 1, typDPT := typDPT);
_MOVE46_OUT := MOVE(EN := M1_001_001_RB601_V.xUpdate_PLC, IN := M1_001_001_RB601_V.xSwitch_OUT, ENO => _MOVE46_ENO);
IF _MOVE46_ENO THEN STLV59_563.STLV59_A_563_001.RB601_V := _MOVE46_OUT; END_IF;
M1_002_001_RB602_V(bPortKNX := 1, dwIndex_DPT := 2, typDPT := typDPT);
_MOVE59_OUT := MOVE(EN := M1_002_001_RB602_V.xUpdate_PLC, IN := M1_002_001_RB602_V.xSwitch_OUT, ENO => _MOVE59_ENO);
IF _MOVE59_ENO THEN STLV59_563.STLV59_A_563_001.RB602_V := _MOVE59_OUT; END_IF;
(* RB603_V *)
(* RB604_V *)
M1_003_001_RB603_V(bPortKNX := 1, dwIndex_DPT := 3, typDPT := typDPT);
_MOVE72_OUT := MOVE(EN := M1_003_001_RB603_V.xUpdate_PLC, IN := M1_003_001_RB603_V.xSwitch_OUT, ENO => _MOVE72_ENO);
IF _MOVE72_ENO THEN STLV59_563.STLV59_A_563_001.RB603_V := _MOVE72_OUT; END_IF;
M1_004_001_RB604_V(bPortKNX := 1, dwIndex_DPT := 4, typDPT := typDPT);
_MOVE85_OUT := MOVE(EN := M1_004_001_RB604_V.xUpdate_PLC, IN := M1_004_001_RB604_V.xSwitch_OUT, ENO => _MOVE85_ENO);
IF _MOVE85_ENO THEN STLV59_563.STLV59_A_563_001.RB604_V := _MOVE85_OUT; END_IF;
(* RB605_V *)
(* RB606_V *)
M1_005_001_RB605_V(bPortKNX := 1, dwIndex_DPT := 5, typDPT := typDPT);
_MOVE98_OUT := MOVE(EN := M1_005_001_RB605_V.xUpdate_PLC, IN := M1_005_001_RB605_V.xSwitch_OUT, ENO => _MOVE98_ENO);
IF _MOVE98_ENO THEN STLV59_563.STLV59_A_563_001.RB605_V := _MOVE98_OUT; END_IF;
M1_006_001_RB606_V(bPortKNX := 1, dwIndex_DPT := 6, typDPT := typDPT);
_MOVE111_OUT := MOVE(EN := M1_006_001_RB606_V.xUpdate_PLC, IN := M1_006_001_RB606_V.xSwitch_OUT, ENO => _MOVE111_ENO);
IF _MOVE111_ENO THEN STLV59_563.STLV59_A_563_001.RB606_V := _MOVE111_OUT; END_IF;
(* RB607_V *)
(* RB608_V *)
M1_007_001_RB607_V(bPortKNX := 1, dwIndex_DPT := 7, typDPT := typDPT);
_MOVE124_OUT := MOVE(EN := M1_007_001_RB607_V.xUpdate_PLC, IN := M1_007_001_RB607_V.xSwitch_OUT, ENO => _MOVE124_ENO);
IF _MOVE124_ENO THEN STLV59_563.STLV59_A_563_001.RB607_V := _MOVE124_OUT; END_IF;
M1_008_001_RB608_V(bPortKNX := 1, dwIndex_DPT := 8, typDPT := typDPT);
_MOVE137_OUT := MOVE(EN := M1_008_001_RB608_V.xUpdate_PLC, IN := M1_008_001_RB608_V.xSwitch_OUT, ENO => _MOVE137_ENO);
IF _MOVE137_ENO THEN STLV59_563.STLV59_A_563_001.RB608_V := _MOVE137_OUT; END_IF;
(* RB609_V *)
(* RB601_HVAC *)
M1_009_001_RB609_V(bPortKNX := 1, dwIndex_DPT := 9, typDPT := typDPT);
_MOVE150_OUT := MOVE(EN := M1_009_001_RB609_V.xUpdate_PLC, IN := M1_009_001_RB609_V.xSwitch_OUT, ENO => _MOVE150_ENO);
IF _MOVE150_ENO THEN STLV59_563.STLV59_A_563_001.RB609_V := _MOVE150_OUT; END_IF;
M1_010_001_RB601_HVAC(bPortKNX := 1, dwIndex_DPT := 10, typDPT := typDPT);
_MOVE163_OUT := MOVE(EN := M1_010_001_RB601_HVAC.xUpdate_PLC, IN := M1_010_001_RB601_HVAC.xSwitch_OUT, ENO => _MOVE163_ENO);
IF _MOVE163_ENO THEN STLV59_563.STLV59_A_563_001.RB601_HVAC := _MOVE163_OUT; END_IF;
(* RB602_HVAC *)
(* RB603_HVAC *)
M1_011_001_RB602_HVAC(bPortKNX := 1, dwIndex_DPT := 11, typDPT := typDPT);
_MOVE176_OUT := MOVE(EN := M1_011_001_RB602_HVAC.xUpdate_PLC, IN := M1_011_001_RB602_HVAC.xSwitch_OUT, ENO => _MOVE176_ENO);
IF _MOVE176_ENO THEN STLV59_563.STLV59_A_563_001.RB602_HVAC := _MOVE176_OUT; END_IF;
M1_012_001_RB603_HVAC(bPortKNX := 1, dwIndex_DPT := 12, typDPT := typDPT);
_MOVE189_OUT := MOVE(EN := M1_012_001_RB603_HVAC.xUpdate_PLC, IN := M1_012_001_RB603_HVAC.xSwitch_OUT, ENO => _MOVE189_ENO);
IF _MOVE189_ENO THEN STLV59_563.STLV59_A_563_001.RB603_HVAC := _MOVE189_OUT; END_IF;
(* RB604_HVAC *)
(* RB605_HVAC *)
M1_013_001_RB604_HVAC(bPortKNX := 1, dwIndex_DPT := 13, typDPT := typDPT);
_MOVE202_OUT := MOVE(EN := M1_013_001_RB604_HVAC.xUpdate_PLC, IN := M1_013_001_RB604_HVAC.xSwitch_OUT, ENO => _MOVE202_ENO);
IF _MOVE202_ENO THEN STLV59_563.STLV59_A_563_001.RB604_HVAC := _MOVE202_OUT; END_IF;
M1_014_001_RB605_HVAC(bPortKNX := 1, dwIndex_DPT := 14, typDPT := typDPT);
_MOVE215_OUT := MOVE(EN := M1_014_001_RB605_HVAC.xUpdate_PLC, IN := M1_014_001_RB605_HVAC.xSwitch_OUT, ENO => _MOVE215_ENO);
IF _MOVE215_ENO THEN STLV59_563.STLV59_A_563_001.RB605_HVAC := _MOVE215_OUT; END_IF;
(* RB606_HVAC *)
(* RB607_HVAC *)
M1_015_001_RB606_HVAC(bPortKNX := 1, dwIndex_DPT := 15, typDPT := typDPT);
_MOVE228_OUT := MOVE(EN := M1_015_001_RB606_HVAC.xUpdate_PLC, IN := M1_015_001_RB606_HVAC.xSwitch_OUT, ENO => _MOVE228_ENO);
IF _MOVE228_ENO THEN STLV59_563.STLV59_A_563_001.RB606_HVAC := _MOVE228_OUT; END_IF;
M1_016_001_RB607_HVAC(bPortKNX := 1, dwIndex_DPT := 16, typDPT := typDPT);
_MOVE241_OUT := MOVE(EN := M1_016_001_RB607_HVAC.xUpdate_PLC, IN := M1_016_001_RB607_HVAC.xSwitch_OUT, ENO => _MOVE241_ENO);
IF _MOVE241_ENO THEN STLV59_563.STLV59_A_563_001.RB607_HVAC := _MOVE241_OUT; END_IF;
(* RB608_HVAC *)
(* RB609_HVAC *)
M1_017_001_RB608_HVAC(bPortKNX := 1, dwIndex_DPT := 17, typDPT := typDPT);
_MOVE254_OUT := MOVE(EN := M1_017_001_RB608_HVAC.xUpdate_PLC, IN := M1_017_001_RB608_HVAC.xSwitch_OUT, ENO => _MOVE254_ENO);
IF _MOVE254_ENO THEN STLV59_563.STLV59_A_563_001.RB608_HVAC := _MOVE254_OUT; END_IF;
M1_018_001_RB609_HVAC(bPortKNX := 1, dwIndex_DPT := 18, typDPT := typDPT);
_MOVE267_OUT := MOVE(EN := M1_018_001_RB609_HVAC.xUpdate_PLC, IN := M1_018_001_RB609_HVAC.xSwitch_OUT, ENO => _MOVE267_ENO);
IF _MOVE267_ENO THEN STLV59_563.STLV59_A_563_001.RB609_HVAC := _MOVE267_OUT; END_IF;
(* RT601_CT *)
(* RT602_CT *)
M1_019_001_RT601_CT(bPortKNX := 1, dwIndex_DPT := 19, typDPT := typDPT);
_MOVE280_OUT := MOVE(EN := M1_019_001_RT601_CT.xUpdate_PLC, IN := M1_019_001_RT601_CT.rValue_OUT, ENO => _MOVE280_ENO);
IF _MOVE280_ENO THEN STLV59_563.STLV59_A_563_001.RT601_CT := _MOVE280_OUT; END_IF;
M1_020_001_RT602_CT(bPortKNX := 1, dwIndex_DPT := 20, typDPT := typDPT);
_MOVE293_OUT := MOVE(EN := M1_020_001_RT602_CT.xUpdate_PLC, IN := M1_020_001_RT602_CT.rValue_OUT, ENO => _MOVE293_ENO);
IF _MOVE293_ENO THEN STLV59_563.STLV59_A_563_001.RT602_CT := _MOVE293_OUT; END_IF;
(* RT603_CT *)
(* RT604_CT *)
M1_021_001_RT603_CT(bPortKNX := 1, dwIndex_DPT := 21, typDPT := typDPT);
_MOVE306_OUT := MOVE(EN := M1_021_001_RT603_CT.xUpdate_PLC, IN := M1_021_001_RT603_CT.rValue_OUT, ENO => _MOVE306_ENO);
IF _MOVE306_ENO THEN STLV59_563.STLV59_A_563_001.RT603_CT := _MOVE306_OUT; END_IF;
M1_022_001_RT604_CT(bPortKNX := 1, dwIndex_DPT := 22, typDPT := typDPT);
_MOVE319_OUT := MOVE(EN := M1_022_001_RT604_CT.xUpdate_PLC, IN := M1_022_001_RT604_CT.rValue_OUT, ENO => _MOVE319_ENO);
IF _MOVE319_ENO THEN STLV59_563.STLV59_A_563_001.RT604_CT := _MOVE319_OUT; END_IF;
(* RT605_CT *)
(* RT606_CT *)
M1_023_001_RT605_CT(bPortKNX := 1, dwIndex_DPT := 23, typDPT := typDPT);
_MOVE332_OUT := MOVE(EN := M1_023_001_RT605_CT.xUpdate_PLC, IN := M1_023_001_RT605_CT.rValue_OUT, ENO => _MOVE332_ENO);
IF _MOVE332_ENO THEN STLV59_563.STLV59_A_563_001.RT605_CT := _MOVE332_OUT; END_IF;
M1_024_001_RT606_CT(bPortKNX := 1, dwIndex_DPT := 24, typDPT := typDPT);
_MOVE345_OUT := MOVE(EN := M1_024_001_RT606_CT.xUpdate_PLC, IN := M1_024_001_RT606_CT.rValue_OUT, ENO => _MOVE345_ENO);
IF _MOVE345_ENO THEN STLV59_563.STLV59_A_563_001.RT606_CT := _MOVE345_OUT; END_IF;
(* RT607_CT *)
(* RT608_CT *)
M1_025_001_RT607_CT(bPortKNX := 1, dwIndex_DPT := 25, typDPT := typDPT);
_MOVE358_OUT := MOVE(EN := M1_025_001_RT607_CT.xUpdate_PLC, IN := M1_025_001_RT607_CT.rValue_OUT, ENO => _MOVE358_ENO);
IF _MOVE358_ENO THEN STLV59_563.STLV59_A_563_001.RT607_CT := _MOVE358_OUT; END_IF;
M1_026_001_RT608_CT(bPortKNX := 1, dwIndex_DPT := 26, typDPT := typDPT);
_MOVE371_OUT := MOVE(EN := M1_026_001_RT608_CT.xUpdate_PLC, IN := M1_026_001_RT608_CT.rValue_OUT, ENO => _MOVE371_ENO);
IF _MOVE371_ENO THEN STLV59_563.STLV59_A_563_001.RT608_CT := _MOVE371_OUT; END_IF;
(* RT609_CT *)
(* RY601_CV *)
M1_027_001_RT609_CT(bPortKNX := 1, dwIndex_DPT := 27, typDPT := typDPT);
_MOVE384_OUT := MOVE(EN := M1_027_001_RT609_CT.xUpdate_PLC, IN := M1_027_001_RT609_CT.rValue_OUT, ENO => _MOVE384_ENO);
IF _MOVE384_ENO THEN STLV59_563.STLV59_A_563_001.RT609_CT := _MOVE384_OUT; END_IF;
M1_028_001_RY601_CV(bPortKNX := 1, dwIndex_DPT := 28, typDPT := typDPT);
_MOVE397_OUT := MOVE(EN := M1_028_001_RY601_CV.xUpdate_PLC, IN := M1_028_001_RY601_CV.rValue_OUT, ENO => _MOVE397_ENO);
IF _MOVE397_ENO THEN STLV59_563.STLV59_A_563_001.RY601_CV := _MOVE397_OUT; END_IF;
(* RY602_CV *)
(* RY603_CV *)
M1_029_001_RY602_CV(bPortKNX := 1, dwIndex_DPT := 29, typDPT := typDPT);
_MOVE410_OUT := MOVE(EN := M1_029_001_RY602_CV.xUpdate_PLC, IN := M1_029_001_RY602_CV.rValue_OUT, ENO => _MOVE410_ENO);
IF _MOVE410_ENO THEN STLV59_563.STLV59_A_563_001.RY602_CV := _MOVE410_OUT; END_IF;
M1_030_001_RY603_CV(bPortKNX := 1, dwIndex_DPT := 30, typDPT := typDPT);
_MOVE423_OUT := MOVE(EN := M1_030_001_RY603_CV.xUpdate_PLC, IN := M1_030_001_RY603_CV.rValue_OUT, ENO => _MOVE423_ENO);
IF _MOVE423_ENO THEN STLV59_563.STLV59_A_563_001.RY603_CV := _MOVE423_OUT; END_IF;
(* RY604_CV *)
(* RY605_CV *)
M1_031_001_RY604_CV(bPortKNX := 1, dwIndex_DPT := 31, typDPT := typDPT);
_MOVE436_OUT := MOVE(EN := M1_031_001_RY604_CV.xUpdate_PLC, IN := M1_031_001_RY604_CV.rValue_OUT, ENO => _MOVE436_ENO);
IF _MOVE436_ENO THEN STLV59_563.STLV59_A_563_001.RY604_CV := _MOVE436_OUT; END_IF;
M1_032_001_RY605_CV(bPortKNX := 1, dwIndex_DPT := 32, typDPT := typDPT);
_MOVE449_OUT := MOVE(EN := M1_032_001_RY605_CV.xUpdate_PLC, IN := M1_032_001_RY605_CV.rValue_OUT, ENO => _MOVE449_ENO);
IF _MOVE449_ENO THEN STLV59_563.STLV59_A_563_001.RY605_CV := _MOVE449_OUT; END_IF;
(* RY606_CV *)
(* RY607_CV *)
M1_033_001_RY606_CV(bPortKNX := 1, dwIndex_DPT := 33, typDPT := typDPT);
_MOVE462_OUT := MOVE(EN := M1_033_001_RY606_CV.xUpdate_PLC, IN := M1_033_001_RY606_CV.rValue_OUT, ENO => _MOVE462_ENO);
IF _MOVE462_ENO THEN STLV59_563.STLV59_A_563_001.RY606_CV := _MOVE462_OUT; END_IF;
M1_034_001_RY607_CV(bPortKNX := 1, dwIndex_DPT := 34, typDPT := typDPT);
_MOVE475_OUT := MOVE(EN := M1_034_001_RY607_CV.xUpdate_PLC, IN := M1_034_001_RY607_CV.rValue_OUT, ENO => _MOVE475_ENO);
IF _MOVE475_ENO THEN STLV59_563.STLV59_A_563_001.RY607_CV := _MOVE475_OUT; END_IF;
(* RY608_CV *)
(* RY609_CV *)
M1_035_001_RY608_CV(bPortKNX := 1, dwIndex_DPT := 35, typDPT := typDPT);
_MOVE488_OUT := MOVE(EN := M1_035_001_RY608_CV.xUpdate_PLC, IN := M1_035_001_RY608_CV.rValue_OUT, ENO => _MOVE488_ENO);
IF _MOVE488_ENO THEN STLV59_563.STLV59_A_563_001.RY608_CV := _MOVE488_OUT; END_IF;
M1_036_001_RY609_CV(bPortKNX := 1, dwIndex_DPT := 36, typDPT := typDPT);
_MOVE501_OUT := MOVE(EN := M1_036_001_RY609_CV.xUpdate_PLC, IN := M1_036_001_RY609_CV.rValue_OUT, ENO => _MOVE501_ENO);
IF _MOVE501_ENO THEN STLV59_563.STLV59_A_563_001.RY609_CV := _MOVE501_OUT; END_IF;
(* LH601_OP *)
(* LH602_OP *)
M1_037_001_LH601_OP(bPortKNX := 1, dwIndex_DPT := 37, rValue_IN := STLV59_563.STLV59_A_563_001.LH601_OP, xUpdate_KNX := i = 0, typDPT := typDPT);
M1_038_001_LH602_OP(bPortKNX := 1, dwIndex_DPT := 38, rValue_IN := STLV59_563.STLV59_A_563_001.LH602_OP, xUpdate_KNX := i = 1, typDPT := typDPT);
(* LH603_OP *)
(* LH604_OP *)
M1_039_001_LH603_OP(bPortKNX := 1, dwIndex_DPT := 39, rValue_IN := STLV59_563.STLV59_A_563_001.LH603_OP, xUpdate_KNX := i = 2, typDPT := typDPT);
M1_040_001_LH604_OP(bPortKNX := 1, dwIndex_DPT := 40, rValue_IN := STLV59_563.STLV59_A_563_001.LH604_OP, xUpdate_KNX := i = 3, typDPT := typDPT);
(* LH605_OP *)
(* LH606_OP *)
M1_041_001_LH605_OP(bPortKNX := 1, dwIndex_DPT := 41, rValue_IN := STLV59_563.STLV59_A_563_001.LH605_OP, xUpdate_KNX := i = 4, typDPT := typDPT);
M1_042_001_LH606_OP(bPortKNX := 1, dwIndex_DPT := 42, rValue_IN := STLV59_563.STLV59_A_563_001.LH606_OP, xUpdate_KNX := i = 5, typDPT := typDPT);
(* LH607_OP *)
(* LH608_OP *)
M1_043_001_LH607_OP(bPortKNX := 1, dwIndex_DPT := 43, rValue_IN := STLV59_563.STLV59_A_563_001.LH607_OP, xUpdate_KNX := i = 6, typDPT := typDPT);
M1_044_001_LH608_OP(bPortKNX := 1, dwIndex_DPT := 44, rValue_IN := STLV59_563.STLV59_A_563_001.LH608_OP, xUpdate_KNX := i = 7, typDPT := typDPT);
(* LH609_OP *)
M1_045_001_LH609_OP(bPortKNX := 1, dwIndex_DPT := 45, rValue_IN := STLV59_563.STLV59_A_563_001.LH609_OP, xUpdate_KNX := i = 8, typDPT := typDPT);
(* Rom 002 *)
(* RB601_V *)
(* RB602_V *)
M1_046_002_RB601_V(bPortKNX := 1, dwIndex_DPT := 46, typDPT := typDPT);
_MOVE659_OUT := MOVE(EN := M1_046_002_RB601_V.xUpdate_PLC, IN := M1_046_002_RB601_V.xSwitch_OUT, ENO => _MOVE659_ENO);
IF _MOVE659_ENO THEN STLV59_563.STLV59_A_563_002.RB601_V := _MOVE659_OUT; END_IF;
M1_047_002_RB602_V(bPortKNX := 1, dwIndex_DPT := 47, typDPT := typDPT);
_MOVE672_OUT := MOVE(EN := M1_047_002_RB602_V.xUpdate_PLC, IN := M1_047_002_RB602_V.xSwitch_OUT, ENO => _MOVE672_ENO);
IF _MOVE672_ENO THEN STLV59_563.STLV59_A_563_002.RB602_V := _MOVE672_OUT; END_IF;
(* RB603_V *)
(* RB604_V *)
M1_048_002_RB603_V(bPortKNX := 1, dwIndex_DPT := 48, typDPT := typDPT);
_MOVE685_OUT := MOVE(EN := M1_048_002_RB603_V.xUpdate_PLC, IN := M1_048_002_RB603_V.xSwitch_OUT, ENO => _MOVE685_ENO);
IF _MOVE685_ENO THEN STLV59_563.STLV59_A_563_002.RB603_V := _MOVE685_OUT; END_IF;
M1_049_002_RB604_V(bPortKNX := 1, dwIndex_DPT := 49, typDPT := typDPT);
_MOVE698_OUT := MOVE(EN := M1_049_002_RB604_V.xUpdate_PLC, IN := M1_049_002_RB604_V.xSwitch_OUT, ENO => _MOVE698_ENO);
IF _MOVE698_ENO THEN STLV59_563.STLV59_A_563_002.RB604_V := _MOVE698_OUT; END_IF;
(* RB605_V *)
(* RB606_V *)
M1_050_002_RB605_V(bPortKNX := 1, dwIndex_DPT := 50, typDPT := typDPT);
_MOVE711_OUT := MOVE(EN := M1_050_002_RB605_V.xUpdate_PLC, IN := M1_050_002_RB605_V.xSwitch_OUT, ENO => _MOVE711_ENO);
IF _MOVE711_ENO THEN STLV59_563.STLV59_A_563_002.RB605_V := _MOVE711_OUT; END_IF;
M1_051_002_RB606_V(bPortKNX := 1, dwIndex_DPT := 51, typDPT := typDPT);
_MOVE724_OUT := MOVE(EN := M1_051_002_RB606_V.xUpdate_PLC, IN := M1_051_002_RB606_V.xSwitch_OUT, ENO => _MOVE724_ENO);
IF _MOVE724_ENO THEN STLV59_563.STLV59_A_563_002.RB606_V := _MOVE724_OUT; END_IF;
(* RB607_V *)
(* RB608_V *)
M1_052_002_RB607_V(bPortKNX := 1, dwIndex_DPT := 52, typDPT := typDPT);
_MOVE737_OUT := MOVE(EN := M1_052_002_RB607_V.xUpdate_PLC, IN := M1_052_002_RB607_V.xSwitch_OUT, ENO => _MOVE737_ENO);
IF _MOVE737_ENO THEN STLV59_563.STLV59_A_563_002.RB607_V := _MOVE737_OUT; END_IF;
M1_053_002_RB608_V(bPortKNX := 1, dwIndex_DPT := 53, typDPT := typDPT);
_MOVE750_OUT := MOVE(EN := M1_053_002_RB608_V.xUpdate_PLC, IN := M1_053_002_RB608_V.xSwitch_OUT, ENO => _MOVE750_ENO);
IF _MOVE750_ENO THEN STLV59_563.STLV59_A_563_002.RB608_V := _MOVE750_OUT; END_IF;
(* RB609_V *)
(* RB601_HVAC *)
M1_054_002_RB609_V(bPortKNX := 1, dwIndex_DPT := 54, typDPT := typDPT);
_MOVE763_OUT := MOVE(EN := M1_054_002_RB609_V.xUpdate_PLC, IN := M1_054_002_RB609_V.xSwitch_OUT, ENO => _MOVE763_ENO);
IF _MOVE763_ENO THEN STLV59_563.STLV59_A_563_002.RB609_V := _MOVE763_OUT; END_IF;
M1_055_002_RB601_HVAC(bPortKNX := 1, dwIndex_DPT := 55, typDPT := typDPT);
_MOVE776_OUT := MOVE(EN := M1_055_002_RB601_HVAC.xUpdate_PLC, IN := M1_055_002_RB601_HVAC.xSwitch_OUT, ENO => _MOVE776_ENO);
IF _MOVE776_ENO THEN STLV59_563.STLV59_A_563_002.RB601_HVAC := _MOVE776_OUT; END_IF;
(* RB602_HVAC *)
(* RB603_HVAC *)
M1_056_002_RB602_HVAC(bPortKNX := 1, dwIndex_DPT := 56, typDPT := typDPT);
_MOVE789_OUT := MOVE(EN := M1_056_002_RB602_HVAC.xUpdate_PLC, IN := M1_056_002_RB602_HVAC.xSwitch_OUT, ENO => _MOVE789_ENO);
IF _MOVE789_ENO THEN STLV59_563.STLV59_A_563_002.RB602_HVAC := _MOVE789_OUT; END_IF;
M1_057_002_RB603_HVAC(bPortKNX := 1, dwIndex_DPT := 57, typDPT := typDPT);
_MOVE802_OUT := MOVE(EN := M1_057_002_RB603_HVAC.xUpdate_PLC, IN := M1_057_002_RB603_HVAC.xSwitch_OUT, ENO => _MOVE802_ENO);
IF _MOVE802_ENO THEN STLV59_563.STLV59_A_563_002.RB603_HVAC := _MOVE802_OUT; END_IF;
(* RB604_HVAC *)
(* RB605_HVAC *)
M1_058_002_RB604_HVAC(bPortKNX := 1, dwIndex_DPT := 58, typDPT := typDPT);
_MOVE815_OUT := MOVE(EN := M1_058_002_RB604_HVAC.xUpdate_PLC, IN := M1_058_002_RB604_HVAC.xSwitch_OUT, ENO => _MOVE815_ENO);
IF _MOVE815_ENO THEN STLV59_563.STLV59_A_563_002.RB604_HVAC := _MOVE815_OUT; END_IF;
M1_059_002_RB605_HVAC(bPortKNX := 1, dwIndex_DPT := 59, typDPT := typDPT);
_MOVE828_OUT := MOVE(EN := M1_059_002_RB605_HVAC.xUpdate_PLC, IN := M1_059_002_RB605_HVAC.xSwitch_OUT, ENO => _MOVE828_ENO);
IF _MOVE828_ENO THEN STLV59_563.STLV59_A_563_002.RB605_HVAC := _MOVE828_OUT; END_IF;
(* RB606_HVAC *)
(* RB607_HVAC *)
M1_060_002_RB606_HVAC(bPortKNX := 1, dwIndex_DPT := 60, typDPT := typDPT);
_MOVE841_OUT := MOVE(EN := M1_060_002_RB606_HVAC.xUpdate_PLC, IN := M1_060_002_RB606_HVAC.xSwitch_OUT, ENO => _MOVE841_ENO);
IF _MOVE841_ENO THEN STLV59_563.STLV59_A_563_002.RB606_HVAC := _MOVE841_OUT; END_IF;
M1_061_002_RB607_HVAC(bPortKNX := 1, dwIndex_DPT := 61, typDPT := typDPT);
_MOVE854_OUT := MOVE(EN := M1_061_002_RB607_HVAC.xUpdate_PLC, IN := M1_061_002_RB607_HVAC.xSwitch_OUT, ENO => _MOVE854_ENO);
IF _MOVE854_ENO THEN STLV59_563.STLV59_A_563_002.RB607_HVAC := _MOVE854_OUT; END_IF;
(* RB608_HVAC *)
(* RB609_HVAC *)
M1_062_002_RB608_HVAC(bPortKNX := 1, dwIndex_DPT := 62, typDPT := typDPT);
_MOVE867_OUT := MOVE(EN := M1_062_002_RB608_HVAC.xUpdate_PLC, IN := M1_062_002_RB608_HVAC.xSwitch_OUT, ENO => _MOVE867_ENO);
IF _MOVE867_ENO THEN STLV59_563.STLV59_A_563_002.RB608_HVAC := _MOVE867_OUT; END_IF;
M1_063_002_RB609_HVAC(bPortKNX := 1, dwIndex_DPT := 63, typDPT := typDPT);
_MOVE880_OUT := MOVE(EN := M1_063_002_RB609_HVAC.xUpdate_PLC, IN := M1_063_002_RB609_HVAC.xSwitch_OUT, ENO => _MOVE880_ENO);
IF _MOVE880_ENO THEN STLV59_563.STLV59_A_563_002.RB609_HVAC := _MOVE880_OUT; END_IF;
(* RT601_CT *)
(* RT602_CT *)
M1_064_002_RT601_CT(bPortKNX := 1, dwIndex_DPT := 64, typDPT := typDPT);
_MOVE893_OUT := MOVE(EN := M1_064_002_RT601_CT.xUpdate_PLC, IN := M1_064_002_RT601_CT.rValue_OUT, ENO => _MOVE893_ENO);
IF _MOVE893_ENO THEN STLV59_563.STLV59_A_563_002.RT601_CT := _MOVE893_OUT; END_IF;
M1_065_002_RT602_CT(bPortKNX := 1, dwIndex_DPT := 65, typDPT := typDPT);
_MOVE906_OUT := MOVE(EN := M1_065_002_RT602_CT.xUpdate_PLC, IN := M1_065_002_RT602_CT.rValue_OUT, ENO => _MOVE906_ENO);
IF _MOVE906_ENO THEN STLV59_563.STLV59_A_563_002.RT602_CT := _MOVE906_OUT; END_IF;
(* RT603_CT *)
(* RT604_CT *)
M1_066_002_RT603_CT(bPortKNX := 1, dwIndex_DPT := 66, typDPT := typDPT);
_MOVE919_OUT := MOVE(EN := M1_066_002_RT603_CT.xUpdate_PLC, IN := M1_066_002_RT603_CT.rValue_OUT, ENO => _MOVE919_ENO);
IF _MOVE919_ENO THEN STLV59_563.STLV59_A_563_002.RT603_CT := _MOVE919_OUT; END_IF;
M1_067_002_RT604_CT(bPortKNX := 1, dwIndex_DPT := 67, typDPT := typDPT);
_MOVE932_OUT := MOVE(EN := M1_067_002_RT604_CT.xUpdate_PLC, IN := M1_067_002_RT604_CT.rValue_OUT, ENO => _MOVE932_ENO);
IF _MOVE932_ENO THEN STLV59_563.STLV59_A_563_002.RT604_CT := _MOVE932_OUT; END_IF;
(* RT605_CT *)
(* RT606_CT *)
M1_068_002_RT605_CT(bPortKNX := 1, dwIndex_DPT := 68, typDPT := typDPT);
_MOVE945_OUT := MOVE(EN := M1_068_002_RT605_CT.xUpdate_PLC, IN := M1_068_002_RT605_CT.rValue_OUT, ENO => _MOVE945_ENO);
IF _MOVE945_ENO THEN STLV59_563.STLV59_A_563_002.RT605_CT := _MOVE945_OUT; END_IF;
M1_069_002_RT606_CT(bPortKNX := 1, dwIndex_DPT := 69, typDPT := typDPT);
_MOVE958_OUT := MOVE(EN := M1_069_002_RT606_CT.xUpdate_PLC, IN := M1_069_002_RT606_CT.rValue_OUT, ENO => _MOVE958_ENO);
IF _MOVE958_ENO THEN STLV59_563.STLV59_A_563_002.RT606_CT := _MOVE958_OUT; END_IF;
(* RT607_CT *)
(* RT608_CT *)
M1_070_002_RT607_CT(bPortKNX := 1, dwIndex_DPT := 70, typDPT := typDPT);
_MOVE971_OUT := MOVE(EN := M1_070_002_RT607_CT.xUpdate_PLC, IN := M1_070_002_RT607_CT.rValue_OUT, ENO => _MOVE971_ENO);
IF _MOVE971_ENO THEN STLV59_563.STLV59_A_563_002.RT607_CT := _MOVE971_OUT; END_IF;
M1_071_002_RT608_CT(bPortKNX := 1, dwIndex_DPT := 71, typDPT := typDPT);
_MOVE984_OUT := MOVE(EN := M1_071_002_RT608_CT.xUpdate_PLC, IN := M1_071_002_RT608_CT.rValue_OUT, ENO => _MOVE984_ENO);
IF _MOVE984_ENO THEN STLV59_563.STLV59_A_563_002.RT608_CT := _MOVE984_OUT; END_IF;
(* RT609_CT *)
(* RY601_CV *)
M1_072_002_RT609_CT(bPortKNX := 1, dwIndex_DPT := 72, typDPT := typDPT);
_MOVE997_OUT := MOVE(EN := M1_072_002_RT609_CT.xUpdate_PLC, IN := M1_072_002_RT609_CT.rValue_OUT, ENO => _MOVE997_ENO);
IF _MOVE997_ENO THEN STLV59_563.STLV59_A_563_002.RT609_CT := _MOVE997_OUT; END_IF;
M1_073_002_RY601_CV(bPortKNX := 1, dwIndex_DPT := 73, typDPT := typDPT);
_MOVE1010_OUT := MOVE(EN := M1_073_002_RY601_CV.xUpdate_PLC, IN := M1_073_002_RY601_CV.rValue_OUT, ENO => _MOVE1010_ENO);
IF _MOVE1010_ENO THEN STLV59_563.STLV59_A_563_002.RY601_CV := _MOVE1010_OUT; END_IF;
(* RY602_CV *)
(* RY603_CV *)
M1_074_002_RY602_CV(bPortKNX := 1, dwIndex_DPT := 74, typDPT := typDPT);
_MOVE1023_OUT := MOVE(EN := M1_074_002_RY602_CV.xUpdate_PLC, IN := M1_074_002_RY602_CV.rValue_OUT, ENO => _MOVE1023_ENO);
IF _MOVE1023_ENO THEN STLV59_563.STLV59_A_563_002.RY602_CV := _MOVE1023_OUT; END_IF;
M1_075_002_RY603_CV(bPortKNX := 1, dwIndex_DPT := 75, typDPT := typDPT);
_MOVE1036_OUT := MOVE(EN := M1_075_002_RY603_CV.xUpdate_PLC, IN := M1_075_002_RY603_CV.rValue_OUT, ENO => _MOVE1036_ENO);
IF _MOVE1036_ENO THEN STLV59_563.STLV59_A_563_002.RY603_CV := _MOVE1036_OUT; END_IF;
(* RY604_CV *)
(* RY605_CV *)
M1_076_002_RY604_CV(bPortKNX := 1, dwIndex_DPT := 76, typDPT := typDPT);
_MOVE1049_OUT := MOVE(EN := M1_076_002_RY604_CV.xUpdate_PLC, IN := M1_076_002_RY604_CV.rValue_OUT, ENO => _MOVE1049_ENO);
IF _MOVE1049_ENO THEN STLV59_563.STLV59_A_563_002.RY604_CV := _MOVE1049_OUT; END_IF;
M1_077_002_RY605_CV(bPortKNX := 1, dwIndex_DPT := 77, typDPT := typDPT);
_MOVE1062_OUT := MOVE(EN := M1_077_002_RY605_CV.xUpdate_PLC, IN := M1_077_002_RY605_CV.rValue_OUT, ENO => _MOVE1062_ENO);
IF _MOVE1062_ENO THEN STLV59_563.STLV59_A_563_002.RY605_CV := _MOVE1062_OUT; END_IF;
(* RY606_CV *)
(* RY607_CV *)
M1_078_002_RY606_CV(bPortKNX := 1, dwIndex_DPT := 78, typDPT := typDPT);
_MOVE1075_OUT := MOVE(EN := M1_078_002_RY606_CV.xUpdate_PLC, IN := M1_078_002_RY606_CV.rValue_OUT, ENO => _MOVE1075_ENO);
IF _MOVE1075_ENO THEN STLV59_563.STLV59_A_563_002.RY606_CV := _MOVE1075_OUT; END_IF;
M1_079_002_RY607_CV(bPortKNX := 1, dwIndex_DPT := 79, typDPT := typDPT);
_MOVE1088_OUT := MOVE(EN := M1_079_002_RY607_CV.xUpdate_PLC, IN := M1_079_002_RY607_CV.rValue_OUT, ENO => _MOVE1088_ENO);
IF _MOVE1088_ENO THEN STLV59_563.STLV59_A_563_002.RY607_CV := _MOVE1088_OUT; END_IF;
(* RY608_CV *)
(* RY609_CV *)
M1_080_002_RY608_CV(bPortKNX := 1, dwIndex_DPT := 80, typDPT := typDPT);
_MOVE1101_OUT := MOVE(EN := M1_080_002_RY608_CV.xUpdate_PLC, IN := M1_080_002_RY608_CV.rValue_OUT, ENO => _MOVE1101_ENO);
IF _MOVE1101_ENO THEN STLV59_563.STLV59_A_563_002.RY608_CV := _MOVE1101_OUT; END_IF;
M1_081_002_RY609_CV(bPortKNX := 1, dwIndex_DPT := 81, typDPT := typDPT);
_MOVE1114_OUT := MOVE(EN := M1_081_002_RY609_CV.xUpdate_PLC, IN := M1_081_002_RY609_CV.rValue_OUT, ENO => _MOVE1114_ENO);
IF _MOVE1114_ENO THEN STLV59_563.STLV59_A_563_002.RY609_CV := _MOVE1114_OUT; END_IF;
(* LH601_OP *)
(* LH602_OP *)
M1_082_002_LH601_OP(bPortKNX := 1, dwIndex_DPT := 82, rValue_IN := STLV59_563.STLV59_A_563_002.LH601_OP, xUpdate_KNX := i = 9, typDPT := typDPT);
M1_083_002_LH602_OP(bPortKNX := 1, dwIndex_DPT := 83, rValue_IN := STLV59_563.STLV59_A_563_002.LH602_OP, xUpdate_KNX := i = 10, typDPT := typDPT);
(* LH603_OP *)
(* LH604_OP *)
M1_084_002_LH603_OP(bPortKNX := 1, dwIndex_DPT := 84, rValue_IN := STLV59_563.STLV59_A_563_002.LH603_OP, xUpdate_KNX := i = 11, typDPT := typDPT);
M1_085_002_LH604_OP(bPortKNX := 1, dwIndex_DPT := 85, rValue_IN := STLV59_563.STLV59_A_563_002.LH604_OP, xUpdate_KNX := i = 12, typDPT := typDPT);
(* LH605_OP *)
(* LH606_OP *)
M1_086_002_LH605_OP(bPortKNX := 1, dwIndex_DPT := 86, rValue_IN := STLV59_563.STLV59_A_563_002.LH605_OP, xUpdate_KNX := i = 13, typDPT := typDPT);
M1_087_002_LH606_OP(bPortKNX := 1, dwIndex_DPT := 87, rValue_IN := STLV59_563.STLV59_A_563_002.LH606_OP, xUpdate_KNX := i = 14, typDPT := typDPT);
(* LH607_OP *)
(* LH608_OP *)
M1_088_002_LH607_OP(bPortKNX := 1, dwIndex_DPT := 88, rValue_IN := STLV59_563.STLV59_A_563_002.LH607_OP, xUpdate_KNX := i = 15, typDPT := typDPT);
M1_089_002_LH608_OP(bPortKNX := 1, dwIndex_DPT := 89, rValue_IN := STLV59_563.STLV59_A_563_002.LH608_OP, xUpdate_KNX := i = 16, typDPT := typDPT);
(* LH609_OP *)
M1_090_002_LH609_OP(bPortKNX := 1, dwIndex_DPT := 90, rValue_IN := STLV59_563.STLV59_A_563_002.LH609_OP, xUpdate_KNX := i = 17, typDPT := typDPT);
(* Rom 003 *)
(* RB601_V *)
(* RB602_V *)
M1_091_003_RB601_V(bPortKNX := 1, dwIndex_DPT := 91, typDPT := typDPT);
_MOVE1272_OUT := MOVE(EN := M1_091_003_RB601_V.xUpdate_PLC, IN := M1_091_003_RB601_V.xSwitch_OUT, ENO => _MOVE1272_ENO);
IF _MOVE1272_ENO THEN STLV59_563.STLV59_A_563_003.RB601_V := _MOVE1272_OUT; END_IF;
M1_092_003_RB602_V(bPortKNX := 1, dwIndex_DPT := 92, typDPT := typDPT);
_MOVE1285_OUT := MOVE(EN := M1_092_003_RB602_V.xUpdate_PLC, IN := M1_092_003_RB602_V.xSwitch_OUT, ENO => _MOVE1285_ENO);
IF _MOVE1285_ENO THEN STLV59_563.STLV59_A_563_003.RB602_V := _MOVE1285_OUT; END_IF;
(* RB603_V *)
(* RB604_V *)
M1_093_003_RB603_V(bPortKNX := 1, dwIndex_DPT := 93, typDPT := typDPT);
_MOVE1298_OUT := MOVE(EN := M1_093_003_RB603_V.xUpdate_PLC, IN := M1_093_003_RB603_V.xSwitch_OUT, ENO => _MOVE1298_ENO);
IF _MOVE1298_ENO THEN STLV59_563.STLV59_A_563_003.RB603_V := _MOVE1298_OUT; END_IF;
M1_094_003_RB604_V(bPortKNX := 1, dwIndex_DPT := 94, typDPT := typDPT);
_MOVE1311_OUT := MOVE(EN := M1_094_003_RB604_V.xUpdate_PLC, IN := M1_094_003_RB604_V.xSwitch_OUT, ENO => _MOVE1311_ENO);
IF _MOVE1311_ENO THEN STLV59_563.STLV59_A_563_003.RB604_V := _MOVE1311_OUT; END_IF;
(* RB605_V *)
(* RB606_V *)
M1_095_003_RB605_V(bPortKNX := 1, dwIndex_DPT := 95, typDPT := typDPT);
_MOVE1324_OUT := MOVE(EN := M1_095_003_RB605_V.xUpdate_PLC, IN := M1_095_003_RB605_V.xSwitch_OUT, ENO => _MOVE1324_ENO);
IF _MOVE1324_ENO THEN STLV59_563.STLV59_A_563_003.RB605_V := _MOVE1324_OUT; END_IF;
M1_096_003_RB606_V(bPortKNX := 1, dwIndex_DPT := 96, typDPT := typDPT);
_MOVE1337_OUT := MOVE(EN := M1_096_003_RB606_V.xUpdate_PLC, IN := M1_096_003_RB606_V.xSwitch_OUT, ENO => _MOVE1337_ENO);
IF _MOVE1337_ENO THEN STLV59_563.STLV59_A_563_003.RB606_V := _MOVE1337_OUT; END_IF;
(* RB607_V *)
(* RB608_V *)
M1_097_003_RB607_V(bPortKNX := 1, dwIndex_DPT := 97, typDPT := typDPT);
_MOVE1350_OUT := MOVE(EN := M1_097_003_RB607_V.xUpdate_PLC, IN := M1_097_003_RB607_V.xSwitch_OUT, ENO => _MOVE1350_ENO);
IF _MOVE1350_ENO THEN STLV59_563.STLV59_A_563_003.RB607_V := _MOVE1350_OUT; END_IF;
M1_098_003_RB608_V(bPortKNX := 1, dwIndex_DPT := 98, typDPT := typDPT);
_MOVE1363_OUT := MOVE(EN := M1_098_003_RB608_V.xUpdate_PLC, IN := M1_098_003_RB608_V.xSwitch_OUT, ENO => _MOVE1363_ENO);
IF _MOVE1363_ENO THEN STLV59_563.STLV59_A_563_003.RB608_V := _MOVE1363_OUT; END_IF;
(* RB609_V *)
(* RB601_HVAC *)
M1_099_003_RB609_V(bPortKNX := 1, dwIndex_DPT := 99, typDPT := typDPT);
_MOVE1376_OUT := MOVE(EN := M1_099_003_RB609_V.xUpdate_PLC, IN := M1_099_003_RB609_V.xSwitch_OUT, ENO => _MOVE1376_ENO);
IF _MOVE1376_ENO THEN STLV59_563.STLV59_A_563_003.RB609_V := _MOVE1376_OUT; END_IF;
M1_100_003_RB601_HVAC(bPortKNX := 1, dwIndex_DPT := 100, typDPT := typDPT);
_MOVE1389_OUT := MOVE(EN := M1_100_003_RB601_HVAC.xUpdate_PLC, IN := M1_100_003_RB601_HVAC.xSwitch_OUT, ENO => _MOVE1389_ENO);
IF _MOVE1389_ENO THEN STLV59_563.STLV59_A_563_003.RB601_HVAC := _MOVE1389_OUT; END_IF;
(* RB602_HVAC *)
(* RB603_HVAC *)
M1_101_003_RB602_HVAC(bPortKNX := 1, dwIndex_DPT := 101, typDPT := typDPT);
_MOVE1402_OUT := MOVE(EN := M1_101_003_RB602_HVAC.xUpdate_PLC, IN := M1_101_003_RB602_HVAC.xSwitch_OUT, ENO => _MOVE1402_ENO);
IF _MOVE1402_ENO THEN STLV59_563.STLV59_A_563_003.RB602_HVAC := _MOVE1402_OUT; END_IF;
M1_102_003_RB603_HVAC(bPortKNX := 1, dwIndex_DPT := 102, typDPT := typDPT);
_MOVE1415_OUT := MOVE(EN := M1_102_003_RB603_HVAC.xUpdate_PLC, IN := M1_102_003_RB603_HVAC.xSwitch_OUT, ENO => _MOVE1415_ENO);
IF _MOVE1415_ENO THEN STLV59_563.STLV59_A_563_003.RB603_HVAC := _MOVE1415_OUT; END_IF;
(* RB604_HVAC *)
(* RB605_HVAC *)
M1_103_003_RB604_HVAC(bPortKNX := 1, dwIndex_DPT := 103, typDPT := typDPT);
_MOVE1428_OUT := MOVE(EN := M1_103_003_RB604_HVAC.xUpdate_PLC, IN := M1_103_003_RB604_HVAC.xSwitch_OUT, ENO => _MOVE1428_ENO);
IF _MOVE1428_ENO THEN STLV59_563.STLV59_A_563_003.RB604_HVAC := _MOVE1428_OUT; END_IF;
M1_104_003_RB605_HVAC(bPortKNX := 1, dwIndex_DPT := 104, typDPT := typDPT);
_MOVE1441_OUT := MOVE(EN := M1_104_003_RB605_HVAC.xUpdate_PLC, IN := M1_104_003_RB605_HVAC.xSwitch_OUT, ENO => _MOVE1441_ENO);
IF _MOVE1441_ENO THEN STLV59_563.STLV59_A_563_003.RB605_HVAC := _MOVE1441_OUT; END_IF;
(* RB606_HVAC *)
(* RB607_HVAC *)
M1_105_003_RB606_HVAC(bPortKNX := 1, dwIndex_DPT := 105, typDPT := typDPT);
_MOVE1454_OUT := MOVE(EN := M1_105_003_RB606_HVAC.xUpdate_PLC, IN := M1_105_003_RB606_HVAC.xSwitch_OUT, ENO => _MOVE1454_ENO);
IF _MOVE1454_ENO THEN STLV59_563.STLV59_A_563_003.RB606_HVAC := _MOVE1454_OUT; END_IF;
M1_106_003_RB607_HVAC(bPortKNX := 1, dwIndex_DPT := 106, typDPT := typDPT);
_MOVE1467_OUT := MOVE(EN := M1_106_003_RB607_HVAC.xUpdate_PLC, IN := M1_106_003_RB607_HVAC.xSwitch_OUT, ENO => _MOVE1467_ENO);
IF _MOVE1467_ENO THEN STLV59_563.STLV59_A_563_003.RB607_HVAC := _MOVE1467_OUT; END_IF;
(* RB608_HVAC *)
(* RB609_HVAC *)
M1_107_003_RB608_HVAC(bPortKNX := 1, dwIndex_DPT := 107, typDPT := typDPT);
_MOVE1480_OUT := MOVE(EN := M1_107_003_RB608_HVAC.xUpdate_PLC, IN := M1_107_003_RB608_HVAC.xSwitch_OUT, ENO => _MOVE1480_ENO);
IF _MOVE1480_ENO THEN STLV59_563.STLV59_A_563_003.RB608_HVAC := _MOVE1480_OUT; END_IF;
M1_108_003_RB609_HVAC(bPortKNX := 1, dwIndex_DPT := 108, typDPT := typDPT);
_MOVE1493_OUT := MOVE(EN := M1_108_003_RB609_HVAC.xUpdate_PLC, IN := M1_108_003_RB609_HVAC.xSwitch_OUT, ENO => _MOVE1493_ENO);
IF _MOVE1493_ENO THEN STLV59_563.STLV59_A_563_003.RB609_HVAC := _MOVE1493_OUT; END_IF;
(* RT601_CT *)
(* RT602_CT *)
M1_109_003_RT601_CT(bPortKNX := 1, dwIndex_DPT := 109, typDPT := typDPT);
_MOVE1506_OUT := MOVE(EN := M1_109_003_RT601_CT.xUpdate_PLC, IN := M1_109_003_RT601_CT.rValue_OUT, ENO => _MOVE1506_ENO);
IF _MOVE1506_ENO THEN STLV59_563.STLV59_A_563_003.RT601_CT := _MOVE1506_OUT; END_IF;
M1_110_003_RT602_CT(bPortKNX := 1, dwIndex_DPT := 110, typDPT := typDPT);
_MOVE1519_OUT := MOVE(EN := M1_110_003_RT602_CT.xUpdate_PLC, IN := M1_110_003_RT602_CT.rValue_OUT, ENO => _MOVE1519_ENO);
IF _MOVE1519_ENO THEN STLV59_563.STLV59_A_563_003.RT602_CT := _MOVE1519_OUT; END_IF;
(* RT603_CT *)
(* RT604_CT *)
M1_111_003_RT603_CT(bPortKNX := 1, dwIndex_DPT := 111, typDPT := typDPT);
_MOVE1532_OUT := MOVE(EN := M1_111_003_RT603_CT.xUpdate_PLC, IN := M1_111_003_RT603_CT.rValue_OUT, ENO => _MOVE1532_ENO);
IF _MOVE1532_ENO THEN STLV59_563.STLV59_A_563_003.RT603_CT := _MOVE1532_OUT; END_IF;
M1_112_003_RT604_CT(bPortKNX := 1, dwIndex_DPT := 112, typDPT := typDPT);
_MOVE1545_OUT := MOVE(EN := M1_112_003_RT604_CT.xUpdate_PLC, IN := M1_112_003_RT604_CT.rValue_OUT, ENO => _MOVE1545_ENO);
IF _MOVE1545_ENO THEN STLV59_563.STLV59_A_563_003.RT604_CT := _MOVE1545_OUT; END_IF;
(* RT605_CT *)
(* RT606_CT *)
M1_113_003_RT605_CT(bPortKNX := 1, dwIndex_DPT := 113, typDPT := typDPT);
_MOVE1558_OUT := MOVE(EN := M1_113_003_RT605_CT.xUpdate_PLC, IN := M1_113_003_RT605_CT.rValue_OUT, ENO => _MOVE1558_ENO);
IF _MOVE1558_ENO THEN STLV59_563.STLV59_A_563_003.RT605_CT := _MOVE1558_OUT; END_IF;
M1_114_003_RT606_CT(bPortKNX := 1, dwIndex_DPT := 114, typDPT := typDPT);
_MOVE1571_OUT := MOVE(EN := M1_114_003_RT606_CT.xUpdate_PLC, IN := M1_114_003_RT606_CT.rValue_OUT, ENO => _MOVE1571_ENO);
IF _MOVE1571_ENO THEN STLV59_563.STLV59_A_563_003.RT606_CT := _MOVE1571_OUT; END_IF;
(* RT607_CT *)
(* RT608_CT *)
M1_115_003_RT607_CT(bPortKNX := 1, dwIndex_DPT := 115, typDPT := typDPT);
_MOVE1584_OUT := MOVE(EN := M1_115_003_RT607_CT.xUpdate_PLC, IN := M1_115_003_RT607_CT.rValue_OUT, ENO => _MOVE1584_ENO);
IF _MOVE1584_ENO THEN STLV59_563.STLV59_A_563_003.RT607_CT := _MOVE1584_OUT; END_IF;
M1_116_003_RT608_CT(bPortKNX := 1, dwIndex_DPT := 116, typDPT := typDPT);
_MOVE1597_OUT := MOVE(EN := M1_116_003_RT608_CT.xUpdate_PLC, IN := M1_116_003_RT608_CT.rValue_OUT, ENO => _MOVE1597_ENO);
IF _MOVE1597_ENO THEN STLV59_563.STLV59_A_563_003.RT608_CT := _MOVE1597_OUT; END_IF;
(* RT609_CT *)
(* RY601_CV *)
M1_117_003_RT609_CT(bPortKNX := 1, dwIndex_DPT := 117, typDPT := typDPT);
_MOVE1610_OUT := MOVE(EN := M1_117_003_RT609_CT.xUpdate_PLC, IN := M1_117_003_RT609_CT.rValue_OUT, ENO => _MOVE1610_ENO);
IF _MOVE1610_ENO THEN STLV59_563.STLV59_A_563_003.RT609_CT := _MOVE1610_OUT; END_IF;
M1_118_003_RY601_CV(bPortKNX := 1, dwIndex_DPT := 118, typDPT := typDPT);
_MOVE1623_OUT := MOVE(EN := M1_118_003_RY601_CV.xUpdate_PLC, IN := M1_118_003_RY601_CV.rValue_OUT, ENO => _MOVE1623_ENO);
IF _MOVE1623_ENO THEN STLV59_563.STLV59_A_563_003.RY601_CV := _MOVE1623_OUT; END_IF;
(* RY602_CV *)
M1_119_003_RY602_CV(bPortKNX := 1, dwIndex_DPT := 119, typDPT := typDPT);
_MOVE1636_OUT := MOVE(EN := M1_119_003_RY602_CV.xUpdate_PLC, IN := M1_119_003_RY602_CV.rValue_OUT, ENO => _MOVE1636_ENO);
IF _MOVE1636_ENO THEN STLV59_563.STLV59_A_563_003.RY602_CV := _MOVE1636_OUT; END_IF;
(* Rom 4K302 *)
(* RB601_V *)
(* RB601_HVAC *)
M1_120_4K302_RB601_V(bPortKNX := 1, dwIndex_DPT := 120, typDPT := typDPT);
_MOVE1650_OUT := MOVE(EN := M1_120_4K302_RB601_V.xUpdate_PLC, IN := M1_120_4K302_RB601_V.xSwitch_OUT, ENO => _MOVE1650_ENO);
IF _MOVE1650_ENO THEN STLV59_563.STLV59_A_563_4K302.RB601_V := _MOVE1650_OUT; END_IF;
M1_121_4K302_RB601_HVAC(bPortKNX := 1, dwIndex_DPT := 121, typDPT := typDPT);
_MOVE1663_OUT := MOVE(EN := M1_121_4K302_RB601_HVAC.xUpdate_PLC, IN := M1_121_4K302_RB601_HVAC.xSwitch_OUT, ENO => _MOVE1663_ENO);
IF _MOVE1663_ENO THEN STLV59_563.STLV59_A_563_4K302.RB601_HVAC := _MOVE1663_OUT; END_IF;
(* RT601_CT *)
(* LH601_CMD *)
M1_122_4K302_RT601_CT(bPortKNX := 1, dwIndex_DPT := 122, typDPT := typDPT);
_MOVE1676_OUT := MOVE(EN := M1_122_4K302_RT601_CT.xUpdate_PLC, IN := M1_122_4K302_RT601_CT.rValue_OUT, ENO => _MOVE1676_ENO);
IF _MOVE1676_ENO THEN STLV59_563.STLV59_A_563_4K302.RT601_CT := _MOVE1676_OUT; END_IF;
M1_123_4K302_LH601_CMD(bPortKNX := 1, dwIndex_DPT := 123, xSwitch_IN := STLV59_563.STLV59_A_563_4K302.LH601_CMD, xUpdate_KNX := i = 18, typDPT := typDPT);
(* Rom 4L302 *)
(* RB601_V *)
(* RB601_HVAC *)
M1_124_4L302_RB601_V(bPortKNX := 1, dwIndex_DPT := 124, typDPT := typDPT);
_MOVE1706_OUT := MOVE(EN := M1_124_4L302_RB601_V.xUpdate_PLC, IN := M1_124_4L302_RB601_V.xSwitch_OUT, ENO => _MOVE1706_ENO);
IF _MOVE1706_ENO THEN STLV59_563.STLV59_A_563_4L302.RB601_V := _MOVE1706_OUT; END_IF;
M1_125_4L302_RB601_HVAC(bPortKNX := 1, dwIndex_DPT := 125, typDPT := typDPT);
_MOVE1719_OUT := MOVE(EN := M1_125_4L302_RB601_HVAC.xUpdate_PLC, IN := M1_125_4L302_RB601_HVAC.xSwitch_OUT, ENO => _MOVE1719_ENO);
IF _MOVE1719_ENO THEN STLV59_563.STLV59_A_563_4L302.RB601_HVAC := _MOVE1719_OUT; END_IF;
(* RT601_CT *)
(* LH601_CMD *)
M1_126_4L302_RT601_CT(bPortKNX := 1, dwIndex_DPT := 126, typDPT := typDPT);
_MOVE1732_OUT := MOVE(EN := M1_126_4L302_RT601_CT.xUpdate_PLC, IN := M1_126_4L302_RT601_CT.rValue_OUT, ENO => _MOVE1732_ENO);
IF _MOVE1732_ENO THEN STLV59_563.STLV59_A_563_4L302.RT601_CT := _MOVE1732_OUT; END_IF;
M1_127_4L302_LH601_CMD(bPortKNX := 1, dwIndex_DPT := 127, xSwitch_IN := STLV59_563.STLV59_A_563_4L302.LH601_CMD, xUpdate_KNX := i = 19, typDPT := typDPT);
(* Rom 4H201 *)
(* RB601_V *)
(* RB601_HVAC *)
M1_128_4H201_RB601_V(bPortKNX := 1, dwIndex_DPT := 128, typDPT := typDPT);
_MOVE1762_OUT := MOVE(EN := M1_128_4H201_RB601_V.xUpdate_PLC, IN := M1_128_4H201_RB601_V.xSwitch_OUT, ENO => _MOVE1762_ENO);
IF _MOVE1762_ENO THEN STLV59_563.STLV59_A_563_4H201.RB601_V := _MOVE1762_OUT; END_IF;
M1_129_4H201_RB601_HVAC(bPortKNX := 1, dwIndex_DPT := 129, typDPT := typDPT);
_MOVE1775_OUT := MOVE(EN := M1_129_4H201_RB601_HVAC.xUpdate_PLC, IN := M1_129_4H201_RB601_HVAC.xSwitch_OUT, ENO => _MOVE1775_ENO);
IF _MOVE1775_ENO THEN STLV59_563.STLV59_A_563_4H201.RB601_HVAC := _MOVE1775_OUT; END_IF;
(* RT601_CT *)
(* RY601_CV *)
M1_130_4H201_RT601_CT(bPortKNX := 1, dwIndex_DPT := 130, typDPT := typDPT);
_MOVE1788_OUT := MOVE(EN := M1_130_4H201_RT601_CT.xUpdate_PLC, IN := M1_130_4H201_RT601_CT.rValue_OUT, ENO => _MOVE1788_ENO);
IF _MOVE1788_ENO THEN STLV59_563.STLV59_A_563_4H201.RT601_CT := _MOVE1788_OUT; END_IF;
M1_131_4H201_RY601_CV(bPortKNX := 1, dwIndex_DPT := 131, typDPT := typDPT);
_MOVE1801_OUT := MOVE(EN := M1_131_4H201_RY601_CV.xUpdate_PLC, IN := M1_131_4H201_RY601_CV.rValue_OUT, ENO => _MOVE1801_ENO);
IF _MOVE1801_ENO THEN STLV59_563.STLV59_A_563_4H201.RY601_CV := _MOVE1801_OUT; END_IF;
(* LH601_OP *)
(* LH601_CMD *)
M1_132_4H201_LH601_OP(bPortKNX := 1, dwIndex_DPT := 132, rValue_IN := STLV59_563.STLV59_A_563_4H201.LH601_OP, xUpdate_KNX := i = 20, typDPT := typDPT);
M1_133_4H201_LH601_CMD(bPortKNX := 1, dwIndex_DPT := 133, xSwitch_IN := STLV59_563.STLV59_A_563_4H201.LH601_CMD, xUpdate_KNX := i = 21, typDPT := typDPT);
(* LC601_OP *)
(* LC601_CMD *)
M1_134_4H201_LC601_OP(bPortKNX := 1, dwIndex_DPT := 134, rValue_IN := STLV59_563.STLV59_A_563_4H201.LC601_OP, xUpdate_KNX := i = 22, typDPT := typDPT);
M1_135_4H201_LC601_CMD(bPortKNX := 1, dwIndex_DPT := 135, xSwitch_IN := STLV59_563.STLV59_A_563_4H201.LC601_CMD, xUpdate_KNX := i = 23, typDPT := typDPT);
(* RT601_SP *)
(* RT601_SP Feedback *)
M1_136_4H201_RT601_SP(bPortKNX := 1, dwIndex_DPT := 136, rValue_IN := STLV59_563.STLV59_A_563_4H201.RT601_SP_D, xUpdate_KNX := NOT STLV59_563.STLV59_A_563_4H201.RB601_HVAC, typDPT := typDPT);
M1_137_4H201_RT601_SP_FB(bPortKNX := 1, dwIndex_DPT := 137, typDPT := typDPT);
_MOVE1890_OUT := MOVE(EN := M1_137_4H201_RT601_SP_FB.xUpdate_PLC, IN := M1_137_4H201_RT601_SP_FB.rValue_OUT, ENO => _MOVE1890_ENO);
IF _MOVE1890_ENO THEN STLV59_563.STLV59_A_563_4H201.RT601_SP_IN := _MOVE1890_OUT; END_IF;
(* LU601_V *)
(* LU601_AL *)
M1_138_4H201_LU601_V(bPortKNX := 1, dwIndex_DPT := 138, typDPT := typDPT);
_MOVE1903_OUT := MOVE(EN := M1_138_4H201_LU601_V.xUpdate_PLC, IN := M1_138_4H201_LU601_V.xSwitch_OUT, ENO => _MOVE1903_ENO);
IF _MOVE1903_ENO THEN STLV59_563.STLV59_A_563_4H201.LU601_V := _MOVE1903_OUT; END_IF;
M1_139_4H201_LU601_AL(bPortKNX := 1, dwIndex_DPT := 139, typDPT := typDPT);
_MOVE1916_OUT := MOVE(EN := M1_139_4H201_LU601_AL.xUpdate_PLC, IN := M1_139_4H201_LU601_AL.xSwitch_OUT, ENO => _MOVE1916_ENO);
IF _MOVE1916_ENO THEN STLV59_563.STLV59_A_563_4H201.LU601_AL := _MOVE1916_OUT; END_IF;
(* LU601_CMD *)
(* OPM_001 *)
M1_140_4H201_LU601_CMD(bPortKNX := 1, dwIndex_DPT := 140, xSwitch_IN := STLV59_563.STLV59_A_563_4H201.LU601_CMD, xUpdate_KNX := i = 24, typDPT := typDPT);
M1_141_4H201_OPM_001(bPortKNX := 1, dwIndex_DPT := 141, bIN := STLV59_563.STLV59_A_563_4H201.OPM_001, xUpdate_KNX := i = 25, typDPT := typDPT);
(* RH601_CV *)
M1_142_4H201_RH601_CV(bPortKNX := 1, dwIndex_DPT := 142, typDPT := typDPT);
_MOVE1961_OUT := MOVE(EN := M1_142_4H201_RH601_CV.xUpdate_PLC, IN := M1_142_4H201_RH601_CV.rValue_OUT, ENO => _MOVE1961_ENO);
IF _MOVE1961_ENO THEN STLV59_563.STLV59_A_563_4H201.RT601_CT := _MOVE1961_OUT; END_IF;
END_PROGRAM

PROGRAM PRG_563_Romstyring
  VAR
    Rom_001 : fbRomtype_99999;  (* 001 *)
    Rom_002 : fbRomtype_99999;  (* 002 *)
    Rom_003 : fbRomtype_9992;  (* 003 *)
    Rom_4K302 : fbRomtype_111001;  (* 4K302 *)
    Rom_4L302 : fbRomtype_111001;  (* 4L302 *)
    Rom_4H201 : fbRomtype_111111111111111;  (* 4H201 *)
  END_VAR

(* CFC diagram, written out as Structured Text *)
(* Rom 001 *)
Rom_001(RB601_HVAC := STLV59_563.STLV59_A_563_001.RB601_HVAC, RB602_HVAC := STLV59_563.STLV59_A_563_001.RB602_HVAC, RB603_HVAC := STLV59_563.STLV59_A_563_001.RB603_HVAC, RB604_HVAC := STLV59_563.STLV59_A_563_001.RB604_HVAC, RB605_HVAC := STLV59_563.STLV59_A_563_001.RB605_HVAC, RB606_HVAC := STLV59_563.STLV59_A_563_001.RB606_HVAC, RB607_HVAC := STLV59_563.STLV59_A_563_001.RB607_HVAC, RB608_HVAC := STLV59_563.STLV59_A_563_001.RB608_HVAC, RB609_HVAC := STLV59_563.STLV59_A_563_001.RB609_HVAC, RT601_CT := STLV59_563.STLV59_A_563_001.RT601_CT, RT602_CT := STLV59_563.STLV59_A_563_001.RT602_CT, RT602_SP := STLV59_563.STLV59_A_563_001.RT602_SP, RT603_CT := STLV59_563.STLV59_A_563_001.RT603_CT, RT603_SP := STLV59_563.STLV59_A_563_001.RT603_SP, RT604_CT := STLV59_563.STLV59_A_563_001.RT604_CT, RT604_SP := STLV59_563.STLV59_A_563_001.RT604_SP, RT605_CT := STLV59_563.STLV59_A_563_001.RT605_CT, RT605_SP := STLV59_563.STLV59_A_563_001.RT605_SP, RT606_CT := STLV59_563.STLV59_A_563_001.RT606_CT, RT606_SP := STLV59_563.STLV59_A_563_001.RT606_SP, RT607_CT := STLV59_563.STLV59_A_563_001.RT607_CT, RT607_SP := STLV59_563.STLV59_A_563_001.RT607_SP, RT608_CT := STLV59_563.STLV59_A_563_001.RT608_CT, RT608_SP := STLV59_563.STLV59_A_563_001.RT608_SP, RT609_CT := STLV59_563.STLV59_A_563_001.RT609_CT, RT609_SP := STLV59_563.STLV59_A_563_001.RT609_SP, RT601_SP_D := STLV59_563.STLV59_A_563_001.RT601_SP_D, RT601_SP_S := STLV59_563.STLV59_A_563_001.RT601_SP_S, RT601_SP_N := STLV59_563.STLV59_A_563_001.RT601_SP_N, RT601_SP_F := STLV59_563.STLV59_A_563_001.RT601_SP_F, OPM := STLV59_563.STLV59_A_563_001.OPM, RY601_CV := STLV59_563.STLV59_A_563_001.RY601_CV, RY602_CV := STLV59_563.STLV59_A_563_001.RY602_CV, RY603_CV := STLV59_563.STLV59_A_563_001.RY603_CV, RY604_CV := STLV59_563.STLV59_A_563_001.RY604_CV, RY605_CV := STLV59_563.STLV59_A_563_001.RY605_CV, RY606_CV := STLV59_563.STLV59_A_563_001.RY606_CV, RY607_CV := STLV59_563.STLV59_A_563_001.RY607_CV, RY608_CV := STLV59_563.STLV59_A_563_001.RY608_CV, RY609_CV := STLV59_563.STLV59_A_563_001.RY609_CV, RY601_SP := STLV59_563.STLV59_A_563_001.RY601_SP, RY601_MAN := STLV59_563.STLV59_A_563_001.RY601_MAN, LH601_MAN := STLV59_563.STLV59_A_563_001.LH601_MAN);
STLV59_563.STLV59_A_563_001.OPM_CV := Rom_001.OPM_CV;
STLV59_563.STLV59_A_563_001.RT601_CS := Rom_001.RT601_CS;
STLV59_563.STLV59_A_563_001.RY601_OP := Rom_001.RY601_OP;
STLV59_563.STLV59_A_563_001.LH601_OP := Rom_001.LH601_OP;
STLV59_563.STLV59_A_563_001.LH602_OP := Rom_001.LH602_OP;
STLV59_563.STLV59_A_563_001.LH603_OP := Rom_001.LH603_OP;
STLV59_563.STLV59_A_563_001.LH604_OP := Rom_001.LH604_OP;
STLV59_563.STLV59_A_563_001.LH605_OP := Rom_001.LH605_OP;
STLV59_563.STLV59_A_563_001.LH606_OP := Rom_001.LH606_OP;
STLV59_563.STLV59_A_563_001.LH607_OP := Rom_001.LH607_OP;
STLV59_563.STLV59_A_563_001.LH608_OP := Rom_001.LH608_OP;
STLV59_563.STLV59_A_563_001.LH609_OP := Rom_001.LH609_OP;
(* Rom 002 *)
Rom_002(RB601_HVAC := STLV59_563.STLV59_A_563_002.RB601_HVAC, RB602_HVAC := STLV59_563.STLV59_A_563_002.RB602_HVAC, RB603_HVAC := STLV59_563.STLV59_A_563_002.RB603_HVAC, RB604_HVAC := STLV59_563.STLV59_A_563_002.RB604_HVAC, RB605_HVAC := STLV59_563.STLV59_A_563_002.RB605_HVAC, RB606_HVAC := STLV59_563.STLV59_A_563_002.RB606_HVAC, RB607_HVAC := STLV59_563.STLV59_A_563_002.RB607_HVAC, RB608_HVAC := STLV59_563.STLV59_A_563_002.RB608_HVAC, RB609_HVAC := STLV59_563.STLV59_A_563_002.RB609_HVAC, RT601_CT := STLV59_563.STLV59_A_563_002.RT601_CT, RT602_CT := STLV59_563.STLV59_A_563_002.RT602_CT, RT602_SP := STLV59_563.STLV59_A_563_002.RT602_SP, RT603_CT := STLV59_563.STLV59_A_563_002.RT603_CT, RT603_SP := STLV59_563.STLV59_A_563_002.RT603_SP, RT604_CT := STLV59_563.STLV59_A_563_002.RT604_CT, RT604_SP := STLV59_563.STLV59_A_563_002.RT604_SP, RT605_CT := STLV59_563.STLV59_A_563_002.RT605_CT, RT605_SP := STLV59_563.STLV59_A_563_002.RT605_SP, RT606_CT := STLV59_563.STLV59_A_563_002.RT606_CT, RT606_SP := STLV59_563.STLV59_A_563_002.RT606_SP, RT607_CT := STLV59_563.STLV59_A_563_002.RT607_CT, RT607_SP := STLV59_563.STLV59_A_563_002.RT607_SP, RT608_CT := STLV59_563.STLV59_A_563_002.RT608_CT, RT608_SP := STLV59_563.STLV59_A_563_002.RT608_SP, RT609_CT := STLV59_563.STLV59_A_563_002.RT609_CT, RT609_SP := STLV59_563.STLV59_A_563_002.RT609_SP, RT601_SP_D := STLV59_563.STLV59_A_563_002.RT601_SP_D, RT601_SP_S := STLV59_563.STLV59_A_563_002.RT601_SP_S, RT601_SP_N := STLV59_563.STLV59_A_563_002.RT601_SP_N, RT601_SP_F := STLV59_563.STLV59_A_563_002.RT601_SP_F, OPM := STLV59_563.STLV59_A_563_002.OPM, RY601_CV := STLV59_563.STLV59_A_563_002.RY601_CV, RY602_CV := STLV59_563.STLV59_A_563_002.RY602_CV, RY603_CV := STLV59_563.STLV59_A_563_002.RY603_CV, RY604_CV := STLV59_563.STLV59_A_563_002.RY604_CV, RY605_CV := STLV59_563.STLV59_A_563_002.RY605_CV, RY606_CV := STLV59_563.STLV59_A_563_002.RY606_CV, RY607_CV := STLV59_563.STLV59_A_563_002.RY607_CV, RY608_CV := STLV59_563.STLV59_A_563_002.RY608_CV, RY609_CV := STLV59_563.STLV59_A_563_002.RY609_CV, RY601_SP := STLV59_563.STLV59_A_563_002.RY601_SP, RY601_MAN := STLV59_563.STLV59_A_563_002.RY601_MAN, LH601_MAN := STLV59_563.STLV59_A_563_002.LH601_MAN);
STLV59_563.STLV59_A_563_002.OPM_CV := Rom_002.OPM_CV;
STLV59_563.STLV59_A_563_002.RT601_CS := Rom_002.RT601_CS;
STLV59_563.STLV59_A_563_002.RY601_OP := Rom_002.RY601_OP;
STLV59_563.STLV59_A_563_002.LH601_OP := Rom_002.LH601_OP;
STLV59_563.STLV59_A_563_002.LH602_OP := Rom_002.LH602_OP;
STLV59_563.STLV59_A_563_002.LH603_OP := Rom_002.LH603_OP;
STLV59_563.STLV59_A_563_002.LH604_OP := Rom_002.LH604_OP;
STLV59_563.STLV59_A_563_002.LH605_OP := Rom_002.LH605_OP;
STLV59_563.STLV59_A_563_002.LH606_OP := Rom_002.LH606_OP;
STLV59_563.STLV59_A_563_002.LH607_OP := Rom_002.LH607_OP;
STLV59_563.STLV59_A_563_002.LH608_OP := Rom_002.LH608_OP;
STLV59_563.STLV59_A_563_002.LH609_OP := Rom_002.LH609_OP;
(* Rom 003 *)
Rom_003(RB601_HVAC := STLV59_563.STLV59_A_563_003.RB601_HVAC, RB602_HVAC := STLV59_563.STLV59_A_563_003.RB602_HVAC, RB603_HVAC := STLV59_563.STLV59_A_563_003.RB603_HVAC, RB604_HVAC := STLV59_563.STLV59_A_563_003.RB604_HVAC, RB605_HVAC := STLV59_563.STLV59_A_563_003.RB605_HVAC, RB606_HVAC := STLV59_563.STLV59_A_563_003.RB606_HVAC, RB607_HVAC := STLV59_563.STLV59_A_563_003.RB607_HVAC, RB608_HVAC := STLV59_563.STLV59_A_563_003.RB608_HVAC, RB609_HVAC := STLV59_563.STLV59_A_563_003.RB609_HVAC, RT601_CT := STLV59_563.STLV59_A_563_003.RT601_CT, RT602_CT := STLV59_563.STLV59_A_563_003.RT602_CT, RT602_SP := STLV59_563.STLV59_A_563_003.RT602_SP, RT603_CT := STLV59_563.STLV59_A_563_003.RT603_CT, RT603_SP := STLV59_563.STLV59_A_563_003.RT603_SP, RT604_CT := STLV59_563.STLV59_A_563_003.RT604_CT, RT604_SP := STLV59_563.STLV59_A_563_003.RT604_SP, RT605_CT := STLV59_563.STLV59_A_563_003.RT605_CT, RT605_SP := STLV59_563.STLV59_A_563_003.RT605_SP, RT606_CT := STLV59_563.STLV59_A_563_003.RT606_CT, RT606_SP := STLV59_563.STLV59_A_563_003.RT606_SP, RT607_CT := STLV59_563.STLV59_A_563_003.RT607_CT, RT607_SP := STLV59_563.STLV59_A_563_003.RT607_SP, RT608_CT := STLV59_563.STLV59_A_563_003.RT608_CT, RT608_SP := STLV59_563.STLV59_A_563_003.RT608_SP, RT609_CT := STLV59_563.STLV59_A_563_003.RT609_CT, RT609_SP := STLV59_563.STLV59_A_563_003.RT609_SP, RT601_SP_D := STLV59_563.STLV59_A_563_003.RT601_SP_D, RT601_SP_S := STLV59_563.STLV59_A_563_003.RT601_SP_S, RT601_SP_N := STLV59_563.STLV59_A_563_003.RT601_SP_N, RT601_SP_F := STLV59_563.STLV59_A_563_003.RT601_SP_F, OPM := STLV59_563.STLV59_A_563_003.OPM, RY601_CV := STLV59_563.STLV59_A_563_003.RY601_CV, RY602_CV := STLV59_563.STLV59_A_563_003.RY602_CV, RY601_SP := STLV59_563.STLV59_A_563_003.RY601_SP, RY601_MAN := STLV59_563.STLV59_A_563_003.RY601_MAN);
STLV59_563.STLV59_A_563_003.OPM_CV := Rom_003.OPM_CV;
STLV59_563.STLV59_A_563_003.RT601_CS := Rom_003.RT601_CS;
STLV59_563.STLV59_A_563_003.RY601_OP := Rom_003.RY601_OP;
(* Rom 4K302 *)
Rom_4K302(RB601_HVAC := STLV59_563.STLV59_A_563_4K302.RB601_HVAC, RT601_CT := STLV59_563.STLV59_A_563_4K302.RT601_CT, RT601_SP_D := STLV59_563.STLV59_A_563_4K302.RT601_SP_D, RT601_SP_S := STLV59_563.STLV59_A_563_4K302.RT601_SP_S, RT601_SP_N := STLV59_563.STLV59_A_563_4K302.RT601_SP_N, RT601_SP_F := STLV59_563.STLV59_A_563_4K302.RT601_SP_F, OPM := STLV59_563.STLV59_A_563_4K302.OPM, LH601_MAN := STLV59_563.STLV59_A_563_4K302.LH601_MAN);
STLV59_563.STLV59_A_563_4K302.OPM_CV := Rom_4K302.OPM_CV;
STLV59_563.STLV59_A_563_4K302.RT601_CS := Rom_4K302.RT601_CS;
STLV59_563.STLV59_A_563_4K302.LH601_CMD := Rom_4K302.LH601_CMD;
(* Rom 4L302 *)
Rom_4L302(RB601_HVAC := STLV59_563.STLV59_A_563_4L302.RB601_HVAC, RT601_CT := STLV59_563.STLV59_A_563_4L302.RT601_CT, RT601_SP_D := STLV59_563.STLV59_A_563_4L302.RT601_SP_D, RT601_SP_S := STLV59_563.STLV59_A_563_4L302.RT601_SP_S, RT601_SP_N := STLV59_563.STLV59_A_563_4L302.RT601_SP_N, RT601_SP_F := STLV59_563.STLV59_A_563_4L302.RT601_SP_F, OPM := STLV59_563.STLV59_A_563_4L302.OPM, LH601_MAN := STLV59_563.STLV59_A_563_4L302.LH601_MAN);
STLV59_563.STLV59_A_563_4L302.OPM_CV := Rom_4L302.OPM_CV;
STLV59_563.STLV59_A_563_4L302.RT601_CS := Rom_4L302.RT601_CS;
STLV59_563.STLV59_A_563_4L302.LH601_CMD := Rom_4L302.LH601_CMD;
(* Rom 4H201 *)
Rom_4H201(RB601_HVAC := STLV59_563.STLV59_A_563_4H201.RB601_HVAC, RT601_CT := STLV59_563.STLV59_A_563_4H201.RT601_CT, RT601_SP_D := STLV59_563.STLV59_A_563_4H201.RT601_SP_D, RT601_SP_S := STLV59_563.STLV59_A_563_4H201.RT601_SP_S, RT601_SP_N := STLV59_563.STLV59_A_563_4H201.RT601_SP_N, RT601_SP_F := STLV59_563.STLV59_A_563_4H201.RT601_SP_F, OPM := STLV59_563.STLV59_A_563_4H201.OPM, RY601_CV := STLV59_563.STLV59_A_563_4H201.RY601_CV, RY601_SP := STLV59_563.STLV59_A_563_4H201.RY601_SP, RY601_MAN := STLV59_563.STLV59_A_563_4H201.RY601_MAN, LH601_MAN := STLV59_563.STLV59_A_563_4H201.LH601_MAN, LC601_SP := STLV59_563.STLV59_A_563_4H201.LC601_SP, LC601_MAN := STLV59_563.STLV59_A_563_4H201.LC601_MAN, RT601_SP_IN := STLV59_563.STLV59_A_563_4H201.RT601_SP_IN, LU601_V := STLV59_563.STLV59_A_563_4H201.LU601_V, RH601_V := STLV59_563.STLV59_A_563_4H201.RH601_CV);
STLV59_563.STLV59_A_563_4H201.OPM_CV := Rom_4H201.OPM_CV;
STLV59_563.STLV59_A_563_4H201.RT601_CS := Rom_4H201.RT601_CS;
STLV59_563.STLV59_A_563_4H201.RY601_OP := Rom_4H201.RY601_OP;
STLV59_563.STLV59_A_563_4H201.LH601_OP := Rom_4H201.LH601_OP;
STLV59_563.STLV59_A_563_4H201.LH601_CMD := Rom_4H201.LH601_CMD;
STLV59_563.STLV59_A_563_4H201.LC601_OP := Rom_4H201.LC601_OP;
STLV59_563.STLV59_A_563_4H201.LC601_CMD := Rom_4H201.LC601_CMD;
STLV59_563.STLV59_A_563_4H201.LU601_CMD := Rom_4H201.LU601_CMD;
STLV59_563.STLV59_A_563_4H201.OPM_001 := Rom_4H201.OPM_001;
END_PROGRAM

PROGRAM PRG_360_HVAC

	STLV59_563.STLV59_A_563_RB001_HVAC:=
(
	STLV59_563.STLV59_A_563_001.RB601_HVAC OR
	STLV59_563.STLV59_A_563_001.RB602_HVAC OR
	STLV59_563.STLV59_A_563_001.RB603_HVAC OR
	STLV59_563.STLV59_A_563_001.RB604_HVAC OR
	STLV59_563.STLV59_A_563_001.RB605_HVAC OR
	STLV59_563.STLV59_A_563_001.RB606_HVAC OR
	STLV59_563.STLV59_A_563_001.RB607_HVAC OR
	STLV59_563.STLV59_A_563_001.RB608_HVAC OR
	STLV59_563.STLV59_A_563_001.RB609_HVAC OR
	STLV59_563.STLV59_A_563_002.RB601_HVAC OR
	STLV59_563.STLV59_A_563_002.RB602_HVAC OR
	STLV59_563.STLV59_A_563_002.RB603_HVAC OR
	STLV59_563.STLV59_A_563_002.RB604_HVAC OR
	STLV59_563.STLV59_A_563_002.RB605_HVAC OR
	STLV59_563.STLV59_A_563_002.RB606_HVAC OR
	STLV59_563.STLV59_A_563_002.RB607_HVAC OR
	STLV59_563.STLV59_A_563_002.RB608_HVAC OR
	STLV59_563.STLV59_A_563_002.RB609_HVAC OR
	STLV59_563.STLV59_A_563_003.RB601_HVAC OR
	STLV59_563.STLV59_A_563_003.RB602_HVAC OR
	STLV59_563.STLV59_A_563_003.RB603_HVAC OR
	STLV59_563.STLV59_A_563_003.RB604_HVAC OR
	STLV59_563.STLV59_A_563_003.RB605_HVAC OR
	STLV59_563.STLV59_A_563_003.RB606_HVAC OR
	STLV59_563.STLV59_A_563_003.RB607_HVAC OR
	STLV59_563.STLV59_A_563_003.RB608_HVAC OR
	STLV59_563.STLV59_A_563_003.RB609_HVAC OR
	STLV59_563.STLV59_A_563_4K302.RB601_HVAC OR
	STLV59_563.STLV59_A_563_4L302.RB601_HVAC OR
	STLV59_563.STLV59_A_563_4H201.RB601_HVAC
);
END_PROGRAM
